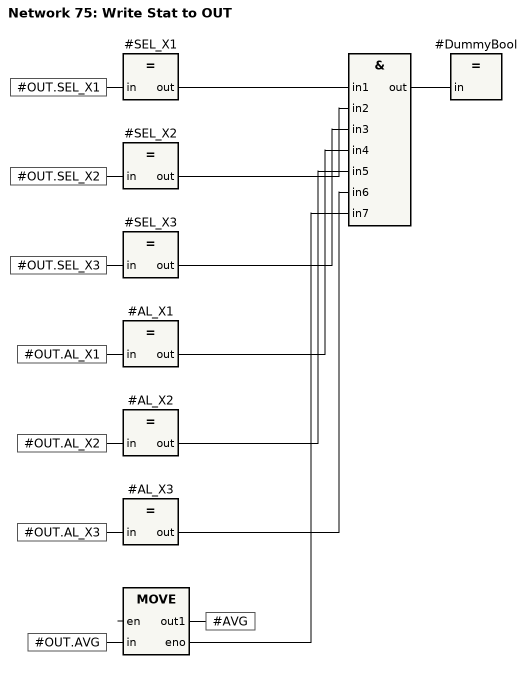
   #SEL_X1 := #OUT.SEL_X1;
   #SEL_X2 := #OUT.SEL_X2;
   #SEL_X3 := #OUT.SEL_X3;
   #AL_X1 := #OUT.AL_X1;
   #AL_X2 := #OUT.AL_X2;
   #AL_X3 := #OUT.AL_X3;
   #AVG := #OUT.AVG;
   #DummyBool := #OUT.SEL_X1 AND #OUT.SEL_X2 AND #OUT.SEL_X3 AND #OUT.AL_X1 AND #OUT.AL_X2 AND #OUT.AL_X3;
END_REGION
END_FUNCTION_BLOCK

FUNCTION_BLOCK "ACESYS_RAMP"   // FB235, FBD
TITLE = ACESYS V8.0 - Build 001 - Ramp Analog Value
{ S7_Optimized_Access := 'FALSE' }
AUTHOR : FLSmidth
FAMILY : ACESYS
NAME : RAMP
VERSION : 8.0
   VAR_INPUT
      Cycle_Time : Int;   // Block Update Time
      SIG_IN : Real;   // Signal Input
      Ramp_Time_Up : Real;   // Ramp Up Time (ms)
      Ramp_Time_Down : Real;   // Ramp Down Time (ms)
      En_Ramp_Up : Bool;   // Enable Ramp Up
      En_Ramp_Down : Bool;   // Enable Ramp Up
   END_VAR
   VAR_OUTPUT
      SIG_OUT : Real;   // Signal Out
   END_VAR
   VAR
      BlockInfo : Struct
         Ace_Version : Int;   // Acesys Block Version Number
         Ace_BuildNo : Int;   // Acesys Block Build Number
         DB_Number : Int;   // Block Instance DB Number
      END_STRUCT;
      Delta_X_Down : Real;   // Number of scan to ramp down
      Delta_X_Up : Real;   // Number of scan to ramp up
      Delta_Y : Real;
      PV_New : Real;
      PV_ToBe : Real;
      ScanTime_Real : Real;
      OUT : Struct
         SIG_OUT : Real;
      END_STRUCT;
      RunTime_Mem : LReal;
      RunTime_RetVal : LReal;
      RunTime_Result : LReal;
   END_VAR
   VAR_TEMP
      Aon : Bool;   // Always ON
      Aoff : Bool;   // Always OFF
      DummyBool : Bool;   // Dummy Bool
      DummyReal : Real;   // Dummy Real
      ScanTime_DINT : DInt;
      SIG_OUT_Internal : Real;   // Signal Out Temp.
      Ramp_Time_Up_Internal : Real;   // Ramp Up Time (ms)
      Ramp_Time_Down_Internal : Real;   // Ramp Down Time (ms)
   END_VAR
   VAR_TEMP   // added for the SCL form of the ladder/FBD networks
      _w1 : Bool;
   END_VAR
BEGIN

REGION Network 1: Always ON
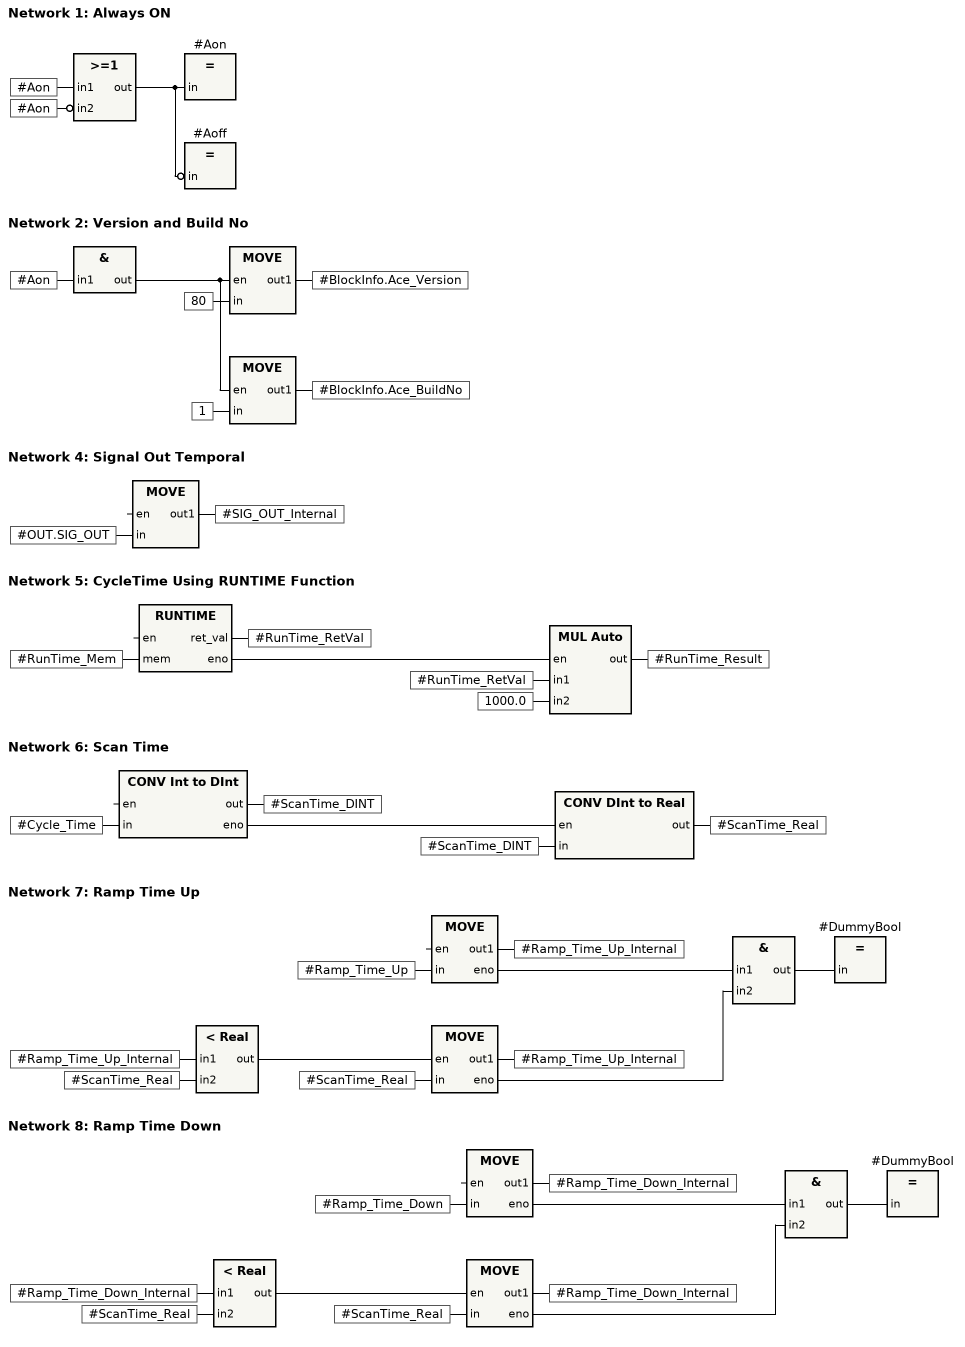
   #Aon := #Aon OR NOT #Aon;
   #Aoff := NOT #Aon;
END_REGION

REGION Network 2: Version and Build No
   IF #Aon THEN
       #BlockInfo.Ace_Version := 80;
       #BlockInfo.Ace_BuildNo := 1;
   END_IF;
END_REGION

REGION Network 3 (STL): Instance DB Number to Faceplate
         L     DINO;
         T     #BlockInfo.DB_Number;
END_REGION

REGION Network 4: Signal Out Temporal
   #SIG_OUT_Internal := #OUT.SIG_OUT;
END_REGION

REGION Network 5: CycleTime Using RUNTIME Function
   // no SCL statement known for Runtime: written as a call
   // ENO of a box is taken as its EN; it also drops when the box reports an error
   #RunTime_RetVal := Runtime(mem := #RunTime_Mem);
   #RunTime_Result := #RunTime_RetVal * 1000.0;
END_REGION

REGION Network 6: Scan Time
   // Build 2 - Cycle_Time added and defined as input to the block instead of MW110
   // ENO of a box is taken as its EN; it also drops when the box reports an error
   #ScanTime_DINT := INT_TO_DINT(#Cycle_Time);
   #ScanTime_Real := DINT_TO_REAL(#ScanTime_DINT);
END_REGION

REGION Network 7: Ramp Time Up
   #Ramp_Time_Up_Internal := #Ramp_Time_Up;
   #_w1 := #Ramp_Time_Up_Internal < #ScanTime_Real;
   IF #_w1 THEN #Ramp_Time_Up_Internal := #ScanTime_Real; END_IF;
   #DummyBool := #_w1;
END_REGION

REGION Network 8: Ramp Time Down
   #Ramp_Time_Down_Internal := #Ramp_Time_Down;
   #_w1 := #Ramp_Time_Down_Internal < #ScanTime_Real;
   IF #_w1 THEN #Ramp_Time_Down_Internal := #ScanTime_Real; END_IF;
   #DummyBool := #_w1;
END_REGION

REGION Network 9: Check for Start Ramping
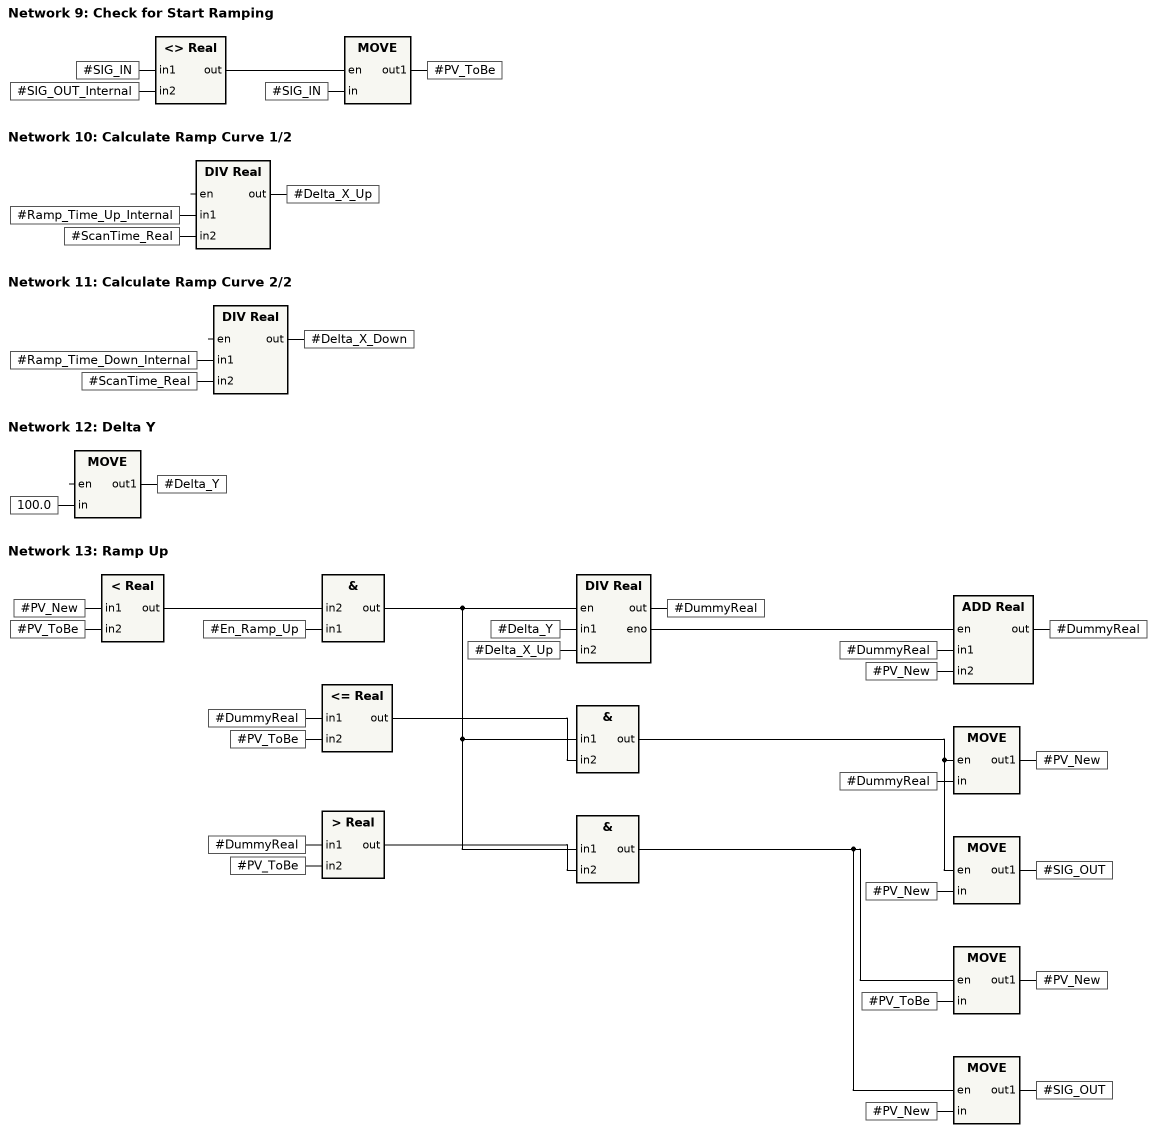
   IF #SIG_IN <> #SIG_OUT_Internal THEN #PV_ToBe := #SIG_IN; END_IF;
END_REGION

REGION Network 10: Calculate Ramp Curve 1/2
   #Delta_X_Up := #Ramp_Time_Up_Internal / #ScanTime_Real;
END_REGION

REGION Network 11: Calculate Ramp Curve 2/2
   #Delta_X_Down := #Ramp_Time_Down_Internal / #ScanTime_Real;
END_REGION

REGION Network 12: Delta Y
   #Delta_Y := 100.0;
END_REGION

REGION Network 13: Ramp Up
   // ENO of a box is taken as its EN; it also drops when the box reports an error
   #_w1 := (#PV_New < #PV_ToBe) AND #En_Ramp_Up;
   IF #_w1 THEN
       #DummyReal := #Delta_Y / #Delta_X_Up;
       #DummyReal := #DummyReal + #PV_New;
   END_IF;
   IF #_w1 AND (#DummyReal <= #PV_ToBe) THEN
       #PV_New := #DummyReal;
       #SIG_OUT := #PV_New;
   END_IF;
   IF #_w1 AND (#DummyReal > #PV_ToBe) THEN
       #PV_New := #PV_ToBe;
       #SIG_OUT := #PV_New;
   END_IF;
END_REGION

REGION Network 14: Ramp Down
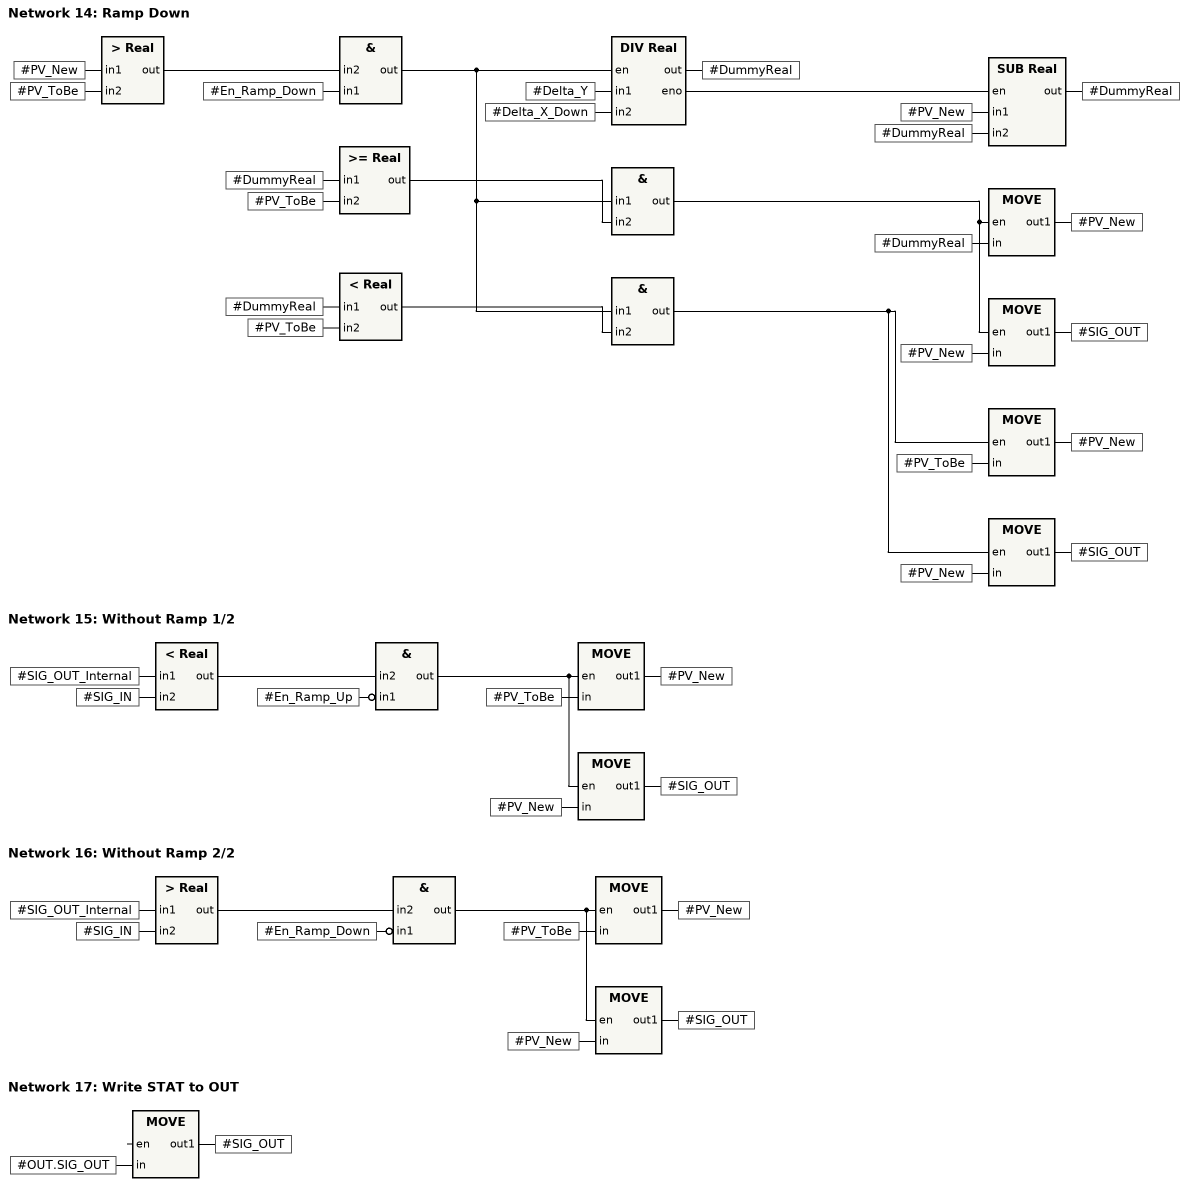
   // ENO of a box is taken as its EN; it also drops when the box reports an error
   #_w1 := (#PV_New > #PV_ToBe) AND #En_Ramp_Down;
   IF #_w1 THEN
       #DummyReal := #Delta_Y / #Delta_X_Down;
       #DummyReal := #PV_New - #DummyReal;
   END_IF;
   IF #_w1 AND (#DummyReal >= #PV_ToBe) THEN
       #PV_New := #DummyReal;
       #SIG_OUT := #PV_New;
   END_IF;
   IF #_w1 AND (#DummyReal < #PV_ToBe) THEN
       #PV_New := #PV_ToBe;
       #SIG_OUT := #PV_New;
   END_IF;
END_REGION

REGION Network 15: Without Ramp 1/2
   IF (#SIG_OUT_Internal < #SIG_IN) AND NOT #En_Ramp_Up THEN
       #PV_New := #PV_ToBe;
       #SIG_OUT := #PV_New;
   END_IF;
END_REGION

REGION Network 16: Without Ramp 2/2
   IF (#SIG_OUT_Internal > #SIG_IN) AND NOT #En_Ramp_Down THEN
       #PV_New := #PV_ToBe;
       #SIG_OUT := #PV_New;
   END_IF;
END_REGION

REGION Network 17: Write STAT to OUT
   #SIG_OUT := #OUT.SIG_OUT;
END_REGION
END_FUNCTION_BLOCK

FUNCTION_BLOCK "ACESTS_RPM"   // FB236, FBD
TITLE = ACESYS V8.0 - Build 005 - RPM Calculation
{ S7_Optimized_Access := 'FALSE' }
AUTHOR : FLSmidth
FAMILY : ACESYS
NAME : RPM
VERSION : 8.0
// Build 003 - Move all elements from TEMP to STAT Area
// Build 004 - RPM_Time Move issue  P_Trig  Placed to last 
// Build 005 - 07 Jan 2021 - Instead of using TIA Runtime Block replaced with Cycle Time Input
   VAR_INPUT
      Cycle_Time : Int;   // Block Update Time
      START : Bool;   // Unit Running
      EN_PULS : Bool;   // Enable Puls Signal
      EN_FREQ : Bool;   // Enable Process Input Signal
      PULS : Bool;   // Puls input
      FREQ : Real;   // Frequence input
      MAX_RPM : Real := 120.0;   // Max RPM (Used to calculate PCT)
      PULS_TURN : Int;   // Puls pr. Revolution
   END_VAR
   VAR_OUTPUT
      OUT_RPM : Real;   // Actual RPM
      OUT_PCT : Real;   // Actual RPM in %
   END_VAR
   VAR
      BlockInfo : Struct
         Ace_Version : Int;   // Acesys Block Version Number
         Ace_BuildNo : Int;   // Acesys Block Build Number
         DB_Number : Int;   // Block Instance DB Number
      END_STRUCT;
      ONS : Struct
         Pulse : Bool;
      END_STRUCT;
      Puls_Turn_Real : Real;
      Max_RPM_Internal : Real;
      PulseTimerAcc : Real;
      RPM_Time : Real;
      OUT_RPM_Temp_1 : Real;
      Out_PCT_Temp_1 : Real;
      TimerAcc : LReal;
      Time_Temp_1 : Int;
      Puls_Turn_Internal : DInt;
      Aon : Bool;
      Aoff : Bool;
      RPM_Pulse : Bool;
      EN_PULS_Temp : Bool;
      EN_FREQ_temp : Bool;
      RunTime_mem : LReal;
      RunTime_RetVal : LReal;
      RunTime_RetVal_Blk : LReal;
      RunTime_Result : LReal;
      OUT : Struct
         OUT_RPM : Real;
         OUT_PCT : Real;
      END_STRUCT;
   END_VAR
   VAR_TEMP
      DummyBool : Bool;
   END_VAR
   VAR_TEMP   // added for the SCL form of the ladder/FBD networks
      _w1 : Bool;
      _w2 : Bool;
   END_VAR
BEGIN

REGION Network 1: Always ON
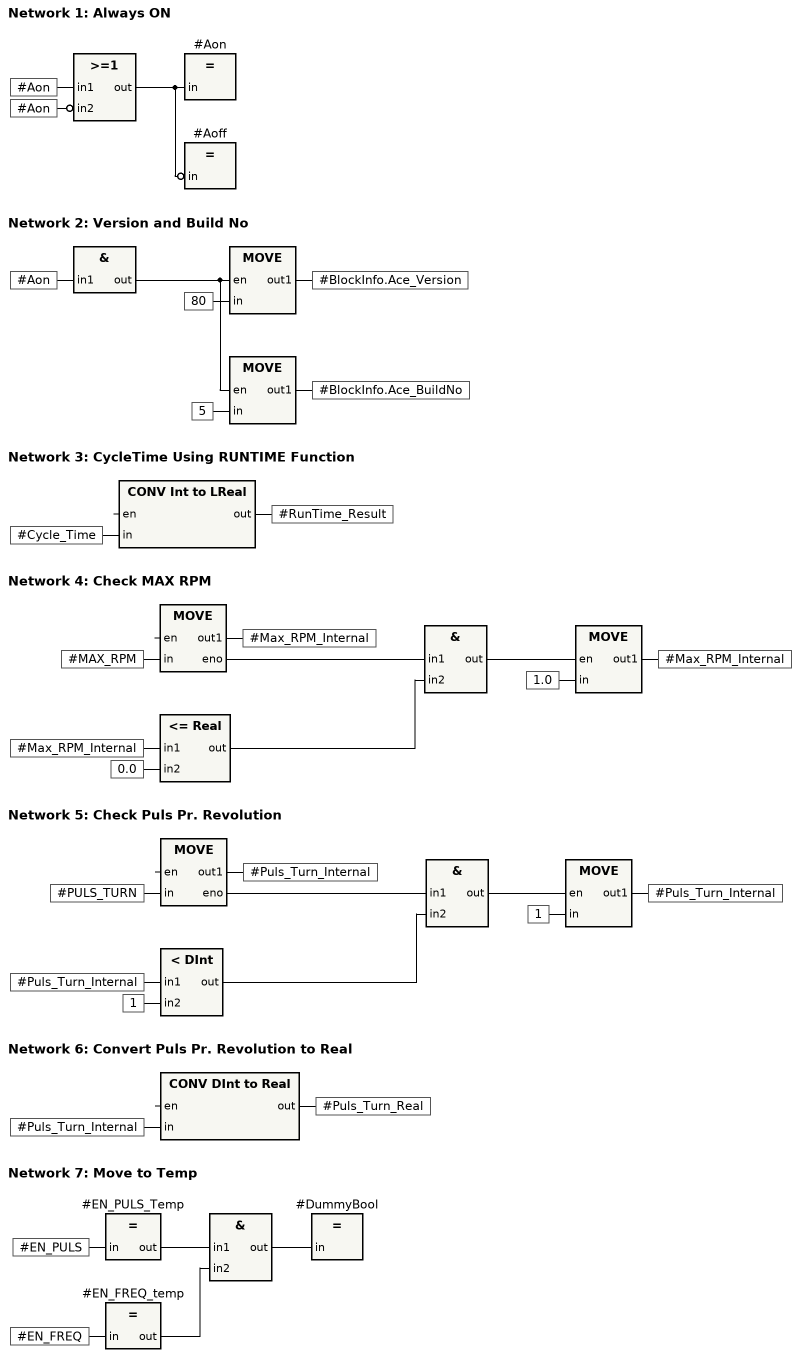
   #Aon := #Aon OR NOT #Aon;
   #Aoff := NOT #Aon;
END_REGION

REGION Network 2: Version and Build No
   IF #Aon THEN
       #BlockInfo.Ace_Version := 80;
       #BlockInfo.Ace_BuildNo := 5;
   END_IF;
END_REGION

REGION Network 3: CycleTime Using RUNTIME Function
   // Build 003 - 27 March 2019 - Use Runtime_RetVal_Blk of second runtime block to accurately get last scan time
   // Build 005 - 07 Jan 2021 - Instead of using TIA Runtime Block Output replaced with Cycle Time Input
   #RunTime_Result := INT_TO_LREAL(#Cycle_Time);
END_REGION

REGION Network 4: Check MAX RPM
   // ENO of a box is taken as its EN; it also drops when the box reports an error
   #Max_RPM_Internal := #MAX_RPM;
   IF #Max_RPM_Internal <= 0.0 THEN #Max_RPM_Internal := 1.0; END_IF;
END_REGION

REGION Network 5: Check Puls Pr. Revolution
   // ENO of a box is taken as its EN; it also drops when the box reports an error
   #Puls_Turn_Internal := #PULS_TURN;
   IF #Puls_Turn_Internal < 1 THEN #Puls_Turn_Internal := 1; END_IF;
END_REGION

REGION Network 6: Convert Puls Pr. Revolution to Real
   #Puls_Turn_Real := DINT_TO_REAL(#Puls_Turn_Internal);
END_REGION

REGION Network 7: Move to Temp
   #EN_PULS_Temp := #EN_PULS;
   #EN_FREQ_temp := #EN_FREQ;
   #DummyBool := #EN_PULS AND #EN_FREQ;
END_REGION

REGION Network 8: Check Configuration
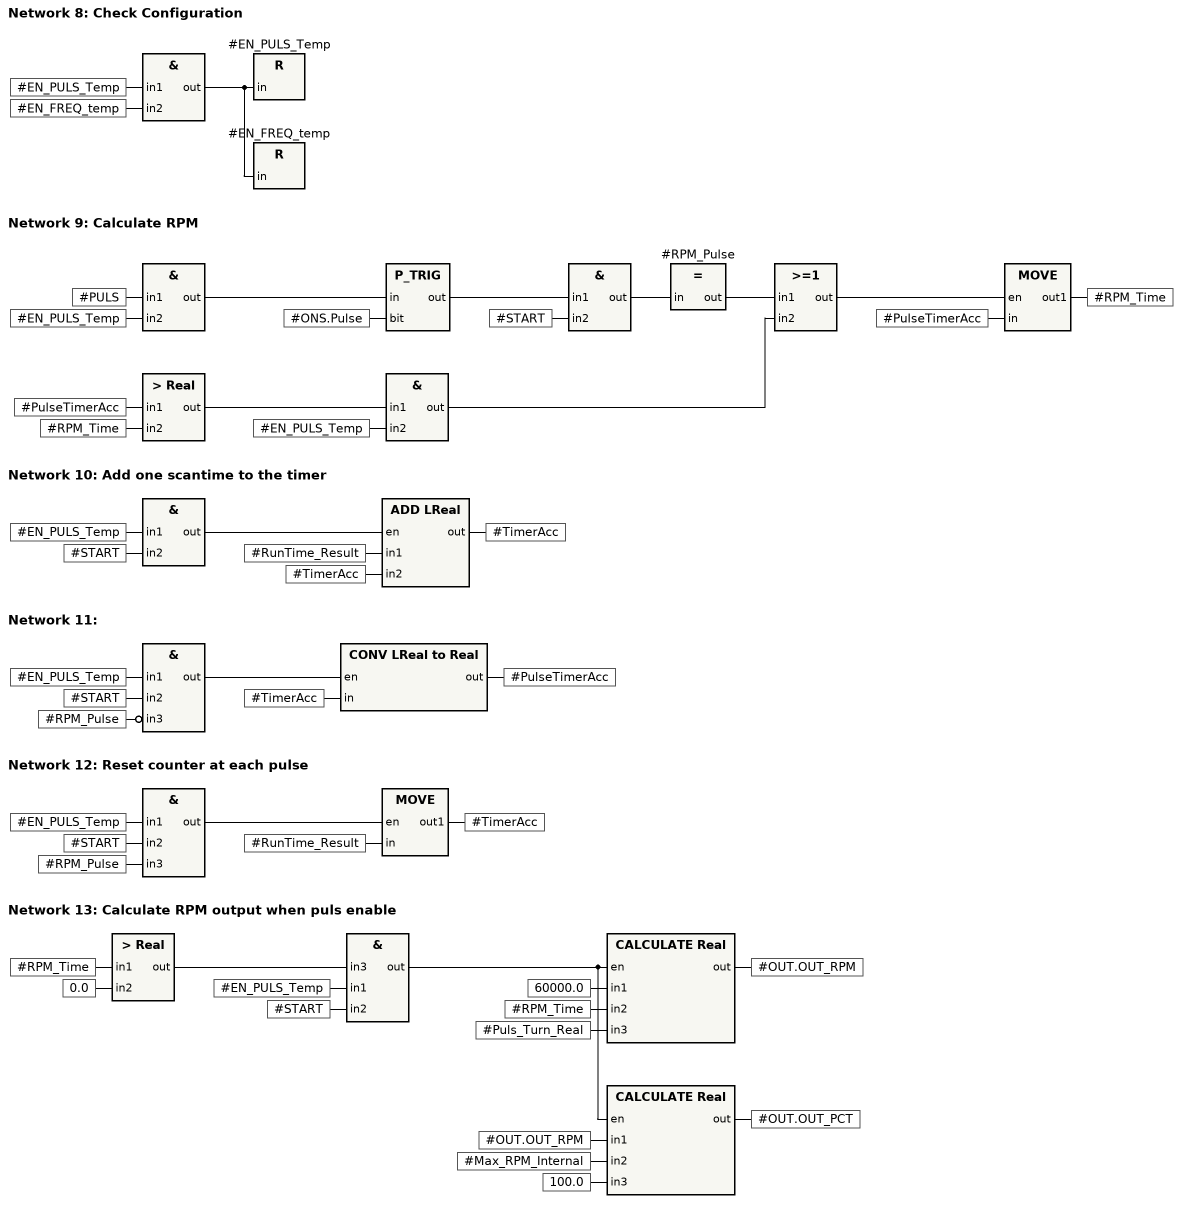
   #_w1 := #EN_PULS_Temp AND #EN_FREQ_temp;
   IF #_w1 THEN
       #EN_PULS_Temp := FALSE;
       #EN_FREQ_temp := FALSE;
   END_IF;
END_REGION

REGION Network 9: Calculate RPM
   // Calculate When a puls or when the time is longer than last Time
   // Build 004 - RPM_Time Move issue - P_Trig  Positioned last
   #_w1 := #PULS AND #EN_PULS_Temp;
   #_w2 := #_w1 AND NOT #ONS.Pulse;   // rising edge
   #ONS.Pulse := #_w1;
   #RPM_Pulse := #_w2 AND #START;
   IF #RPM_Pulse OR ((#PulseTimerAcc > #RPM_Time) AND #EN_PULS_Temp) THEN
       #RPM_Time := #PulseTimerAcc;
   END_IF;
END_REGION

REGION Network 10: Add one scantime to the timer
   // Build 003 - 27 March 2019 - Replace CycleTIme with Runtime_Result for internal Scan time of FB
   IF #EN_PULS_Temp AND #START THEN #TimerAcc := #RunTime_Result + #TimerAcc; END_IF;
END_REGION

REGION Network 11
   IF #EN_PULS_Temp AND #START AND NOT #RPM_Pulse THEN #PulseTimerAcc := LREAL_TO_REAL(#TimerAcc); END_IF;
END_REGION

REGION Network 12: Reset counter at each pulse
   // Build 003 - 27 March 2019 - Replace CycleTIme with Runtime_Result for internal Scan time of FB
   IF #EN_PULS_Temp AND #START AND #RPM_Pulse THEN #TimerAcc := #RunTime_Result; END_IF;
END_REGION

REGION Network 13: Calculate RPM output when puls enable
   // Build 005 - Average PCT Logic Typo Recified,Added 100.0 as IN3
   IF (#RPM_Time > 0.0) AND #EN_PULS_Temp AND #START THEN
       #OUT.OUT_RPM := (60000.0/#RPM_Time/#Puls_Turn_Real);
       #OUT.OUT_PCT := (#OUT.OUT_RPM/#Max_RPM_Internal)*100.0;
   END_IF;
END_REGION

REGION Network 14: Calculate RPM (Analog)
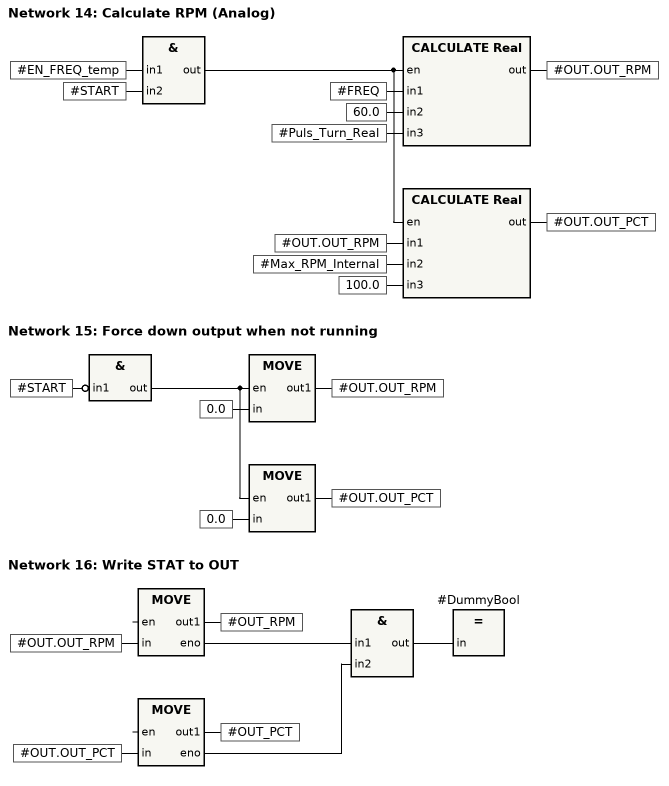
   IF #EN_FREQ_temp AND #START THEN
       #OUT.OUT_RPM := (#FREQ*60.0)/#Puls_Turn_Real;
       #OUT.OUT_PCT := (#OUT.OUT_RPM/#Max_RPM_Internal)*100.0;
   END_IF;
END_REGION

REGION Network 15: Force down output when not running
   IF NOT #START THEN
       #OUT.OUT_RPM := 0.0;
       #OUT.OUT_PCT := 0.0;
   END_IF;
END_REGION

REGION Network 16: Write STAT to OUT
   #OUT_RPM := #OUT.OUT_RPM;
   #OUT_PCT := #OUT.OUT_PCT;
   #DummyBool := TRUE;
END_REGION

REGION Network 17: Runtime Calculation of the block
   // Build 003 - 27 March 2019 - New Network - Runtime Block added to last network to accurately read FB execution time
   // Build 005 - 07 Jan 2021 - TIA Runtime Instruction deleted, Replace with Cycle Time Input
END_REGION
END_FUNCTION_BLOCK

FUNCTION_BLOCK "ACESYS_POWER"   // FB237, FBD
TITLE = ACESYS V8.0 - Build 001 - POWER MONITORING
{ S7_Optimized_Access := 'FALSE' }
AUTHOR : FLSmidth
FAMILY : ACESYS
NAME : POWER
VERSION : 8.0
   VAR_INPUT
      AL_SUPR : Bool;   // Alarm Supress by Program
   END_VAR
   VAR_OUTPUT
      MSW : "ACESYS_HMI_STAT_32T";
   END_VAR
   VAR_IN_OUT
      TOKEN : "ACESYS_TOKEN";
   END_VAR
   VAR
      BlockInfo : Struct
         Ace_Version : Int;   // Acesys Block Version Number
         Ace_BuildNo : Int;   // Acesys Block Build Number
         DB_Number : Int;   // Block Instance DB Number
      END_STRUCT;
      FP_CMD : Struct
         Spare_08 : Bool;
         Spare_09 : Bool;
         Spare_10 : Bool;
         Spare_11 : Bool;
         Spare_12 : Bool;
         Spare_13 : Bool;
         Spare_14 : Bool;
         AckAlarm : Bool;
         Reset : Bool;
         Spare_01 : Bool;
         Spare_02 : Bool;
         Spare_03 : Bool;
         Spare_04 : Bool;
         Spare_05 : Bool;
         Spare_06 : Bool;
         Spare_07 : Bool;
      END_STRUCT;
      FP_SEL : Struct
         Spare_08 : Bool;
         Spare_09 : Bool;
         Spare_10 : Bool;
         Spare_11 : Bool;
         Spare_12 : Bool;
         Spare_13 : Bool;
         Spare_14 : Bool;
         Spare_15 : Bool;
         Type_Monitor : Bool;
         Type_MVfeeder : Bool;
         Type_MVmotor : Bool;
         Type_NotSelected : Bool;
         ParentSupress : Bool;
         ParentSupressUnit : Bool;
         Spare_06 : Bool;
         Spare_07 : Bool;
      END_STRUCT;
      FP_SHOW : Struct
         VOLT_LNPH : Bool;   // Phase to pahse & Line to Neutral Voltage V/kV)
         CURR_LN : Bool;   // Line Current
         APOW_PH : Bool;   // Phase Power kW/MW)
         FRQ : Bool;   // Frequency (Hz)
         APOW_AVG : Bool;   // Average Apparent Power (kVA/MVA)
         RTPOW_AVG : Bool;   // Average Reactive Power (kW/MW)
         VOLT_UNBAL : Bool;   // Voltage Unbalance (%)
         CURR_UNBAL : Bool;   // Current unbalance (%)
         VOLT_THD : Bool;   // Total Hormonic Distorsion Voltage (%)
         CURR_THD : Bool;   // Total Hormonic Distorsion Current (%)
         RENG : Bool;   // Average Reactive Energy (kVARH/MVARH)
         kWH_REV : Bool;   // Reverse kWH (kWhr/MWhr)
         kVAH_FwdRev : Bool;   // kVAH Forward/Reverse(kVAH/MVAH)
         kVARH_Rev : Bool;   // kVARH Reverse(kVARH/MVARH)
         MD_kW_Fwd : Bool;   // kW Forward (kW/MW)
         MD_kW_Rev : Bool;   // kW Reverse (kW/MW)
         MD_kVAr_Fwd : Bool;   // kVA Forward (kVAr/MVAr)
         MD_kVAr_Rev : Bool;   // kVA Reverse (kVAr/MVAr)
         HORM_5TH : Bool;   // 5th Order Hormonics
         HORM_7TH : Bool;   // 7th Order Hormonics
         HORM_11TH : Bool;   // 11th Order Hormonics
         MWT : Bool;   // Motor Winding temperature
         MBT : Bool;   // Motor Bearing temperature
         TWT : Bool;   // Transformer Winding temperature
         TOT : Bool;   // Transformer Oil temperature
         RunHrs : Bool;   // Run Hours
         PB_Reset : Bool;
         PQ2 : Bool;   // Power Quality 2 Group Box
         Temperature : Bool;   // Power Group Box
         Spare19 : Bool;   // Energy Group Box
         Spare18 : Bool;
         Spare17 : Bool;
         Spare16 : Bool;
         Spare15 : Bool;
         Spare14 : Bool;
         Spare13 : Bool;
         Spare12 : Bool;
         Spare11 : Bool;
         Spare10 : Bool;
         Spare09 : Bool;
         Spare08 : Bool;
         Spare07 : Bool;
         Spare06 : Bool;
         Spare05 : Bool;
         Spare04 : Bool;
         Spare03 : Bool;
         Spare02 : Bool;
         Spare01 : Bool;
      END_STRUCT;
      FP_VIS : Struct
         VOLT_LNPH : Bool;   // Phase to pahse & Line to Neutral Voltage V/kV)
         CURR_LN : Bool;   // Line Current
         APOW_PH : Bool;   // Phase Power kW/MW)
         FRQ : Bool;   // Frequency (Hz)
         APOW_AVG : Bool;   // Average Apparent Power (kVA/MVA)
         RTPOW_AVG : Bool;   // Average Reactive Power (kW/MW)
         VOLT_UNBAL : Bool;   // Voltage Unbalance (%)
         CURR_UNBAL : Bool;   // Current unbalance (%)
         VOLT_THD : Bool;   // Total Hormonic Distorsion Voltage (%)
         CURR_THD : Bool;   // Total Hormonic Distorsion Current (%)
         RENG : Bool;   // Average Reactive Energy (kVARH/MVARH)
         kWH_REV : Bool;   // Reverse kWH (kWhr/MWhr)
         kVAH_FwdRev : Bool;   // kVAH Forward/Reverse(kVAH/MVAH)
         kVARH_Rev : Bool;   // kVARH Reverse(kVARH/MVARH)
         MD_kW_Fwd : Bool;   // kW Forward (kW/MW)
         MD_kW_Rev : Bool;   // kW Reverse (kW/MW)
         MD_kVAr_Fwd : Bool;   // kVA Forward (kVAr/MVAr)
         MD_kVAr_Rev : Bool;   // kVA Reverse (kVAr/MVAr)
         HORM_5TH : Bool;   // 5th Order Hormonics
         HORM_7TH : Bool;   // 7th Order Hormonics
         HORM_11TH : Bool;   // 11th Order Hormonics
         MWT : Bool;   // Motor Winding temperature
         MBT : Bool;   // Motor Bearing temperature
         TWT : Bool;   // Transformer Winding temperature
         TOT : Bool;   // Transformer Oil temperature
         RunHrs : Bool;   // Run Hours
         PB_Reset : Bool;   // Show Push Button Reset
         PQ2 : Bool;   // Power Quality 2 Group Box
         Power : Bool;   // Power Group Box
         Energy : Bool;   // Energy Group Box
         Temperature : Bool;
         Spare17 : Bool;
         Spare16 : Bool;
         Spare15 : Bool;
         Spare14 : Bool;
         Spare13 : Bool;
         Spare12 : Bool;
         Spare11 : Bool;
         Spare10 : Bool;
         Spare09 : Bool;
         Spare08 : Bool;
         Spare07 : Bool;
         Spare06 : Bool;
         Spare05 : Bool;
         Spare04 : Bool;
         Spare03 : Bool;
         Spare02 : Bool;
         Spare01 : Bool;
      END_STRUCT;
      LINK : "ACESYS_PowerLink";
      Volt_L1N : Real;   // R Phase to Neutral Voltage Calc
      Volt_L2N : Real;   // Y Phase to Neutral Voltage Calc
      Volt_L3N : Real;   // B Phase to Neutral Voltage Calc
      ONS : Struct
         Spare_08 : Bool;
         Spare_09 : Bool;
         Spare_10 : Bool;
         Spare_11 : Bool;
         Spare_12 : Bool;
         Spare_13 : Bool;
         Spare_14 : Bool;
         Spare_15 : Bool;
         AckAlarm : Bool;
         Spare_01 : Bool;
         Spare_02 : Bool;
         Spare_03 : Bool;
         Spare_04 : Bool;
         Spare_05 : Bool;
         Spare_06 : Bool;
         Spare_07 : Bool;
      END_STRUCT;
      StatusWork : Int;
      AlarmNo : Int;
      AlarmNo_Old : Int;
      CMD_Reset : Bool;
      CMD_AckAlarm : Bool;
      ALARM_SupressionActive : Bool;
      ALARM_AlarmPresent : Bool;
      ALARM_FailureAckRequired : Bool;
      FPCMD_RESET_TMR : TON_TIME;
      MSW_Status_Trans : Int;
   END_VAR
   VAR_TEMP
      ADAPT_Pntr : Struct
         DB_Number : Word;
         Offset_Address : DWord;
      END_STRUCT;
      Aon : Bool;
      Aoff : Bool;
      DummyBool : Bool;
      DummyInt : Int;
      DummyDInt : DInt;
      Temp_AR1 : DWord;
      TEMP_AR2 : DWord;
      Offset : DWord;
      Pntr_ADAPT : ANY;
      Pntr_ADAPT_LC : ANY;
      Pntr_DATA : ANY;
      Pntr_ADAPT_Source : ANY;
   END_VAR
   VAR_TEMP   // added for the SCL form of the ladder/FBD networks
      _w1 : Bool;
   END_VAR
BEGIN

REGION Network 1: Always ON
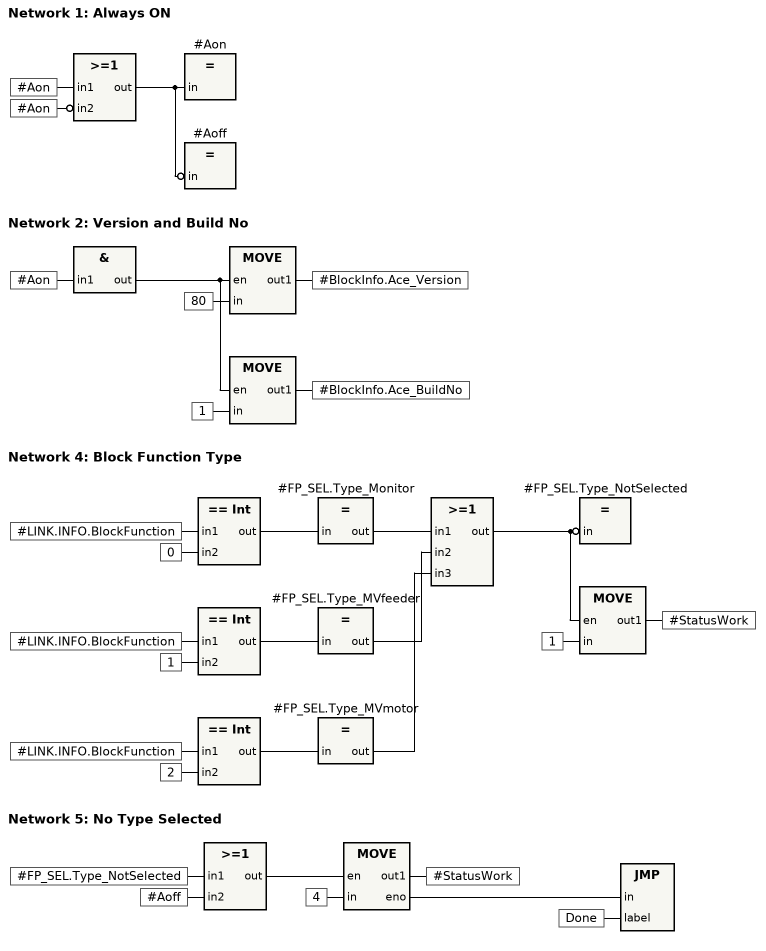
   #Aon := #Aon OR NOT #Aon;
   #Aoff := NOT #Aon;
END_REGION

REGION Network 2: Version and Build No
   IF #Aon THEN
       #BlockInfo.Ace_Version := 80;
       #BlockInfo.Ace_BuildNo := 1;
   END_IF;
END_REGION

REGION Network 3 (STL): Instance DB Number to Faceplate
         L     DINO;
         T     #BlockInfo.DB_Number;
END_REGION

REGION Network 4: Block Function Type
   #FP_SEL.Type_Monitor := #LINK.INFO.BlockFunction = 0;
   #FP_SEL.Type_MVfeeder := #LINK.INFO.BlockFunction = 1;
   #FP_SEL.Type_MVmotor := #LINK.INFO.BlockFunction = 2;
   #_w1 := #FP_SEL.Type_Monitor OR #FP_SEL.Type_MVfeeder OR #FP_SEL.Type_MVmotor;
   #FP_SEL.Type_NotSelected := NOT #_w1;
   IF #_w1 THEN #StatusWork := 1; END_IF;
END_REGION

REGION Network 5: No Type Selected
   // ENO of a box is taken as its EN; it also drops when the box reports an error
   #_w1 := #FP_SEL.Type_NotSelected OR #Aoff;
   IF #_w1 THEN
       #StatusWork := 4;
       GOTO Done;
   END_IF;
END_REGION

REGION Network 6: Set Show Parameters
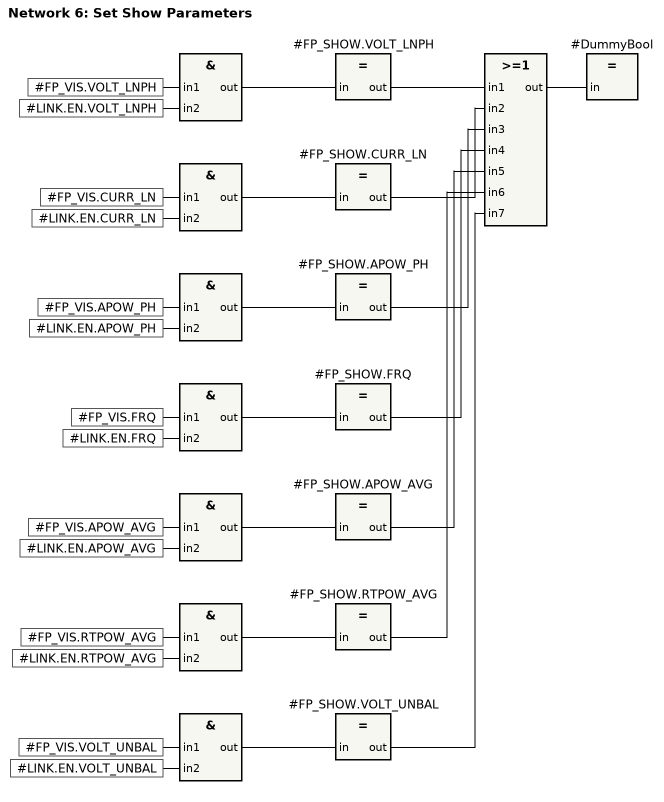
   #FP_SHOW.VOLT_LNPH := #FP_VIS.VOLT_LNPH AND #LINK.EN.VOLT_LNPH;
   #FP_SHOW.CURR_LN := #FP_VIS.CURR_LN AND #LINK.EN.CURR_LN;
   #FP_SHOW.APOW_PH := #FP_VIS.APOW_PH AND #LINK.EN.APOW_PH;
   #FP_SHOW.FRQ := #FP_VIS.FRQ AND #LINK.EN.FRQ;
   #FP_SHOW.APOW_AVG := #FP_VIS.APOW_AVG AND #LINK.EN.APOW_AVG;
   #FP_SHOW.RTPOW_AVG := #FP_VIS.RTPOW_AVG AND #LINK.EN.RTPOW_AVG;
   #FP_SHOW.VOLT_UNBAL := #FP_VIS.VOLT_UNBAL AND #LINK.EN.VOLT_UNBAL;
   #DummyBool := #FP_SHOW.VOLT_LNPH OR #FP_SHOW.CURR_LN OR #FP_SHOW.APOW_PH OR #FP_SHOW.FRQ OR #FP_SHOW.APOW_AVG OR #FP_SHOW.RTPOW_AVG OR #FP_SHOW.VOLT_UNBAL;
END_REGION

REGION Network 7: Set Show Parameters
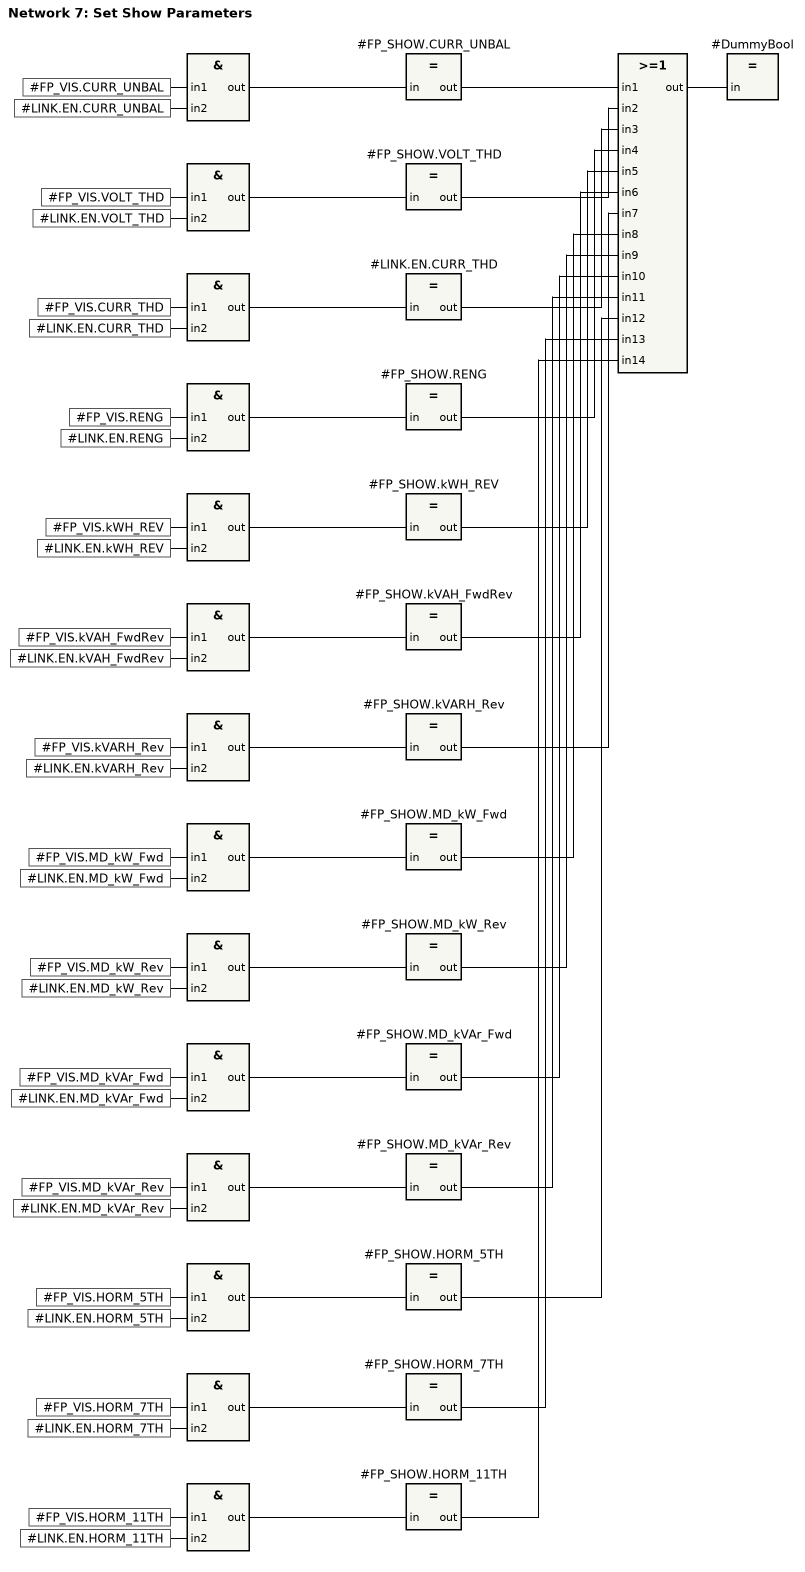
   #FP_SHOW.CURR_UNBAL := #FP_VIS.CURR_UNBAL AND #LINK.EN.CURR_UNBAL;
   #FP_SHOW.VOLT_THD := #FP_VIS.VOLT_THD AND #LINK.EN.VOLT_THD;
   #LINK.EN.CURR_THD := #FP_VIS.CURR_THD AND #LINK.EN.CURR_THD;
   #FP_SHOW.RENG := #FP_VIS.RENG AND #LINK.EN.RENG;
   #FP_SHOW.kWH_REV := #FP_VIS.kWH_REV AND #LINK.EN.kWH_REV;
   #FP_SHOW.kVAH_FwdRev := #FP_VIS.kVAH_FwdRev AND #LINK.EN.kVAH_FwdRev;
   #FP_SHOW.kVARH_Rev := #FP_VIS.kVARH_Rev AND #LINK.EN.kVARH_Rev;
   #FP_SHOW.MD_kW_Fwd := #FP_VIS.MD_kW_Fwd AND #LINK.EN.MD_kW_Fwd;
   #FP_SHOW.MD_kW_Rev := #FP_VIS.MD_kW_Rev AND #LINK.EN.MD_kW_Rev;
   #FP_SHOW.MD_kVAr_Fwd := #FP_VIS.MD_kVAr_Fwd AND #LINK.EN.MD_kVAr_Fwd;
   #FP_SHOW.MD_kVAr_Rev := #FP_VIS.MD_kVAr_Rev AND #LINK.EN.MD_kVAr_Rev;
   #FP_SHOW.HORM_5TH := #FP_VIS.HORM_5TH AND #LINK.EN.HORM_5TH;
   #FP_SHOW.HORM_7TH := #FP_VIS.HORM_7TH AND #LINK.EN.HORM_7TH;
   #FP_SHOW.HORM_11TH := #FP_VIS.HORM_11TH AND #LINK.EN.HORM_11TH;
   #DummyBool := #FP_SHOW.CURR_UNBAL OR #FP_SHOW.VOLT_THD OR #LINK.EN.CURR_THD OR #FP_SHOW.RENG OR #FP_SHOW.kWH_REV OR #FP_SHOW.kVAH_FwdRev OR #FP_SHOW.kVARH_Rev OR #FP_SHOW.MD_kW_Fwd OR #FP_SHOW.MD_kW_Rev OR #FP_SHOW.MD_kVAr_Fwd OR #FP_SHOW.MD_kVAr_Rev OR #FP_SHOW.HORM_5TH OR #FP_SHOW.HORM_7TH OR #FP_SHOW.HORM_11TH;
END_REGION

REGION Network 8: Set Show Parameters
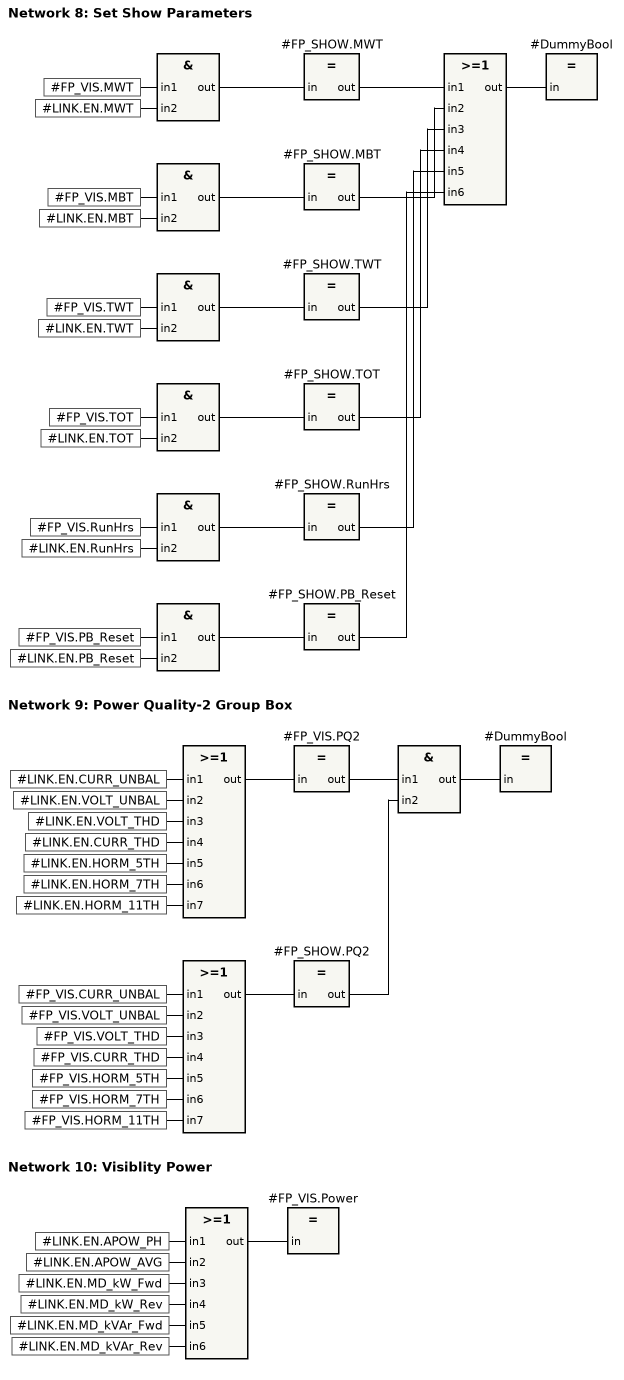
   #FP_SHOW.MWT := #FP_VIS.MWT AND #LINK.EN.MWT;
   #FP_SHOW.MBT := #FP_VIS.MBT AND #LINK.EN.MBT;
   #FP_SHOW.TWT := #FP_VIS.TWT AND #LINK.EN.TWT;
   #FP_SHOW.TOT := #FP_VIS.TOT AND #LINK.EN.TOT;
   #FP_SHOW.RunHrs := #FP_VIS.RunHrs AND #LINK.EN.RunHrs;
   #FP_SHOW.PB_Reset := #FP_VIS.PB_Reset AND #LINK.EN.PB_Reset;
   #DummyBool := #FP_SHOW.MWT OR #FP_SHOW.MBT OR #FP_SHOW.TWT OR #FP_SHOW.TOT OR #FP_SHOW.RunHrs OR #FP_SHOW.PB_Reset;
END_REGION

REGION Network 9: Power Quality-2 Group Box
   #FP_VIS.PQ2 := #LINK.EN.CURR_UNBAL OR #LINK.EN.VOLT_UNBAL OR #LINK.EN.VOLT_THD OR #LINK.EN.CURR_THD OR #LINK.EN.HORM_5TH OR #LINK.EN.HORM_7TH OR #LINK.EN.HORM_11TH;
   #FP_SHOW.PQ2 := #FP_VIS.CURR_UNBAL OR #FP_VIS.VOLT_UNBAL OR #FP_VIS.VOLT_THD OR #FP_VIS.CURR_THD OR #FP_VIS.HORM_5TH OR #FP_VIS.HORM_7TH OR #FP_VIS.HORM_11TH;
   #DummyBool := #FP_VIS.PQ2 AND #FP_SHOW.PQ2;
END_REGION

REGION Network 10: Visiblity Power
   #FP_VIS.Power := #LINK.EN.APOW_PH OR #LINK.EN.APOW_AVG OR #LINK.EN.MD_kW_Fwd OR #LINK.EN.MD_kW_Rev OR #LINK.EN.MD_kVAr_Fwd OR #LINK.EN.MD_kVAr_Rev;
END_REGION

REGION Network 11: Visiblity Energy
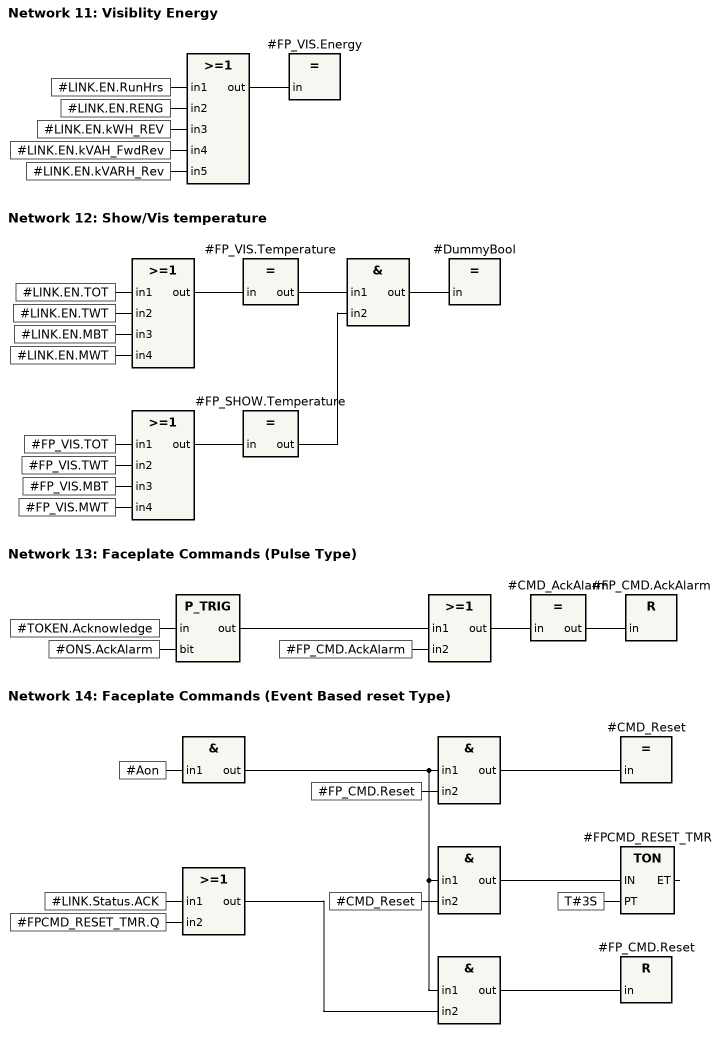
   #FP_VIS.Energy := #LINK.EN.RunHrs OR #LINK.EN.RENG OR #LINK.EN.kWH_REV OR #LINK.EN.kVAH_FwdRev OR #LINK.EN.kVARH_Rev;
END_REGION

REGION Network 12: Show/Vis temperature
   #FP_VIS.Temperature := #LINK.EN.TOT OR #LINK.EN.TWT OR #LINK.EN.MBT OR #LINK.EN.MWT;
   #FP_SHOW.Temperature := #FP_VIS.TOT OR #FP_VIS.TWT OR #FP_VIS.MBT OR #FP_VIS.MWT;
   #DummyBool := #FP_VIS.Temperature AND #FP_SHOW.Temperature;
END_REGION

REGION Network 13: Faceplate Commands (Pulse Type)
   #_w1 := #TOKEN.Acknowledge AND NOT #ONS.AckAlarm;   // rising edge
   #ONS.AckAlarm := #TOKEN.Acknowledge;
   #CMD_AckAlarm := #_w1 OR #FP_CMD.AckAlarm;
   IF #CMD_AckAlarm THEN #FP_CMD.AckAlarm := FALSE; END_IF;
END_REGION

REGION Network 14: Faceplate Commands (Event Based reset Type)
   #CMD_Reset := #Aon AND #FP_CMD.Reset;
   #FPCMD_RESET_TMR(IN := #Aon AND #CMD_Reset, PT := T#3S);   // TON
   IF #Aon AND (#LINK.Status.ACK OR #FPCMD_RESET_TMR.Q) THEN #FP_CMD.Reset := FALSE; END_IF;
END_REGION

REGION Network 15: Phase to Neutral Voltage Calcuation
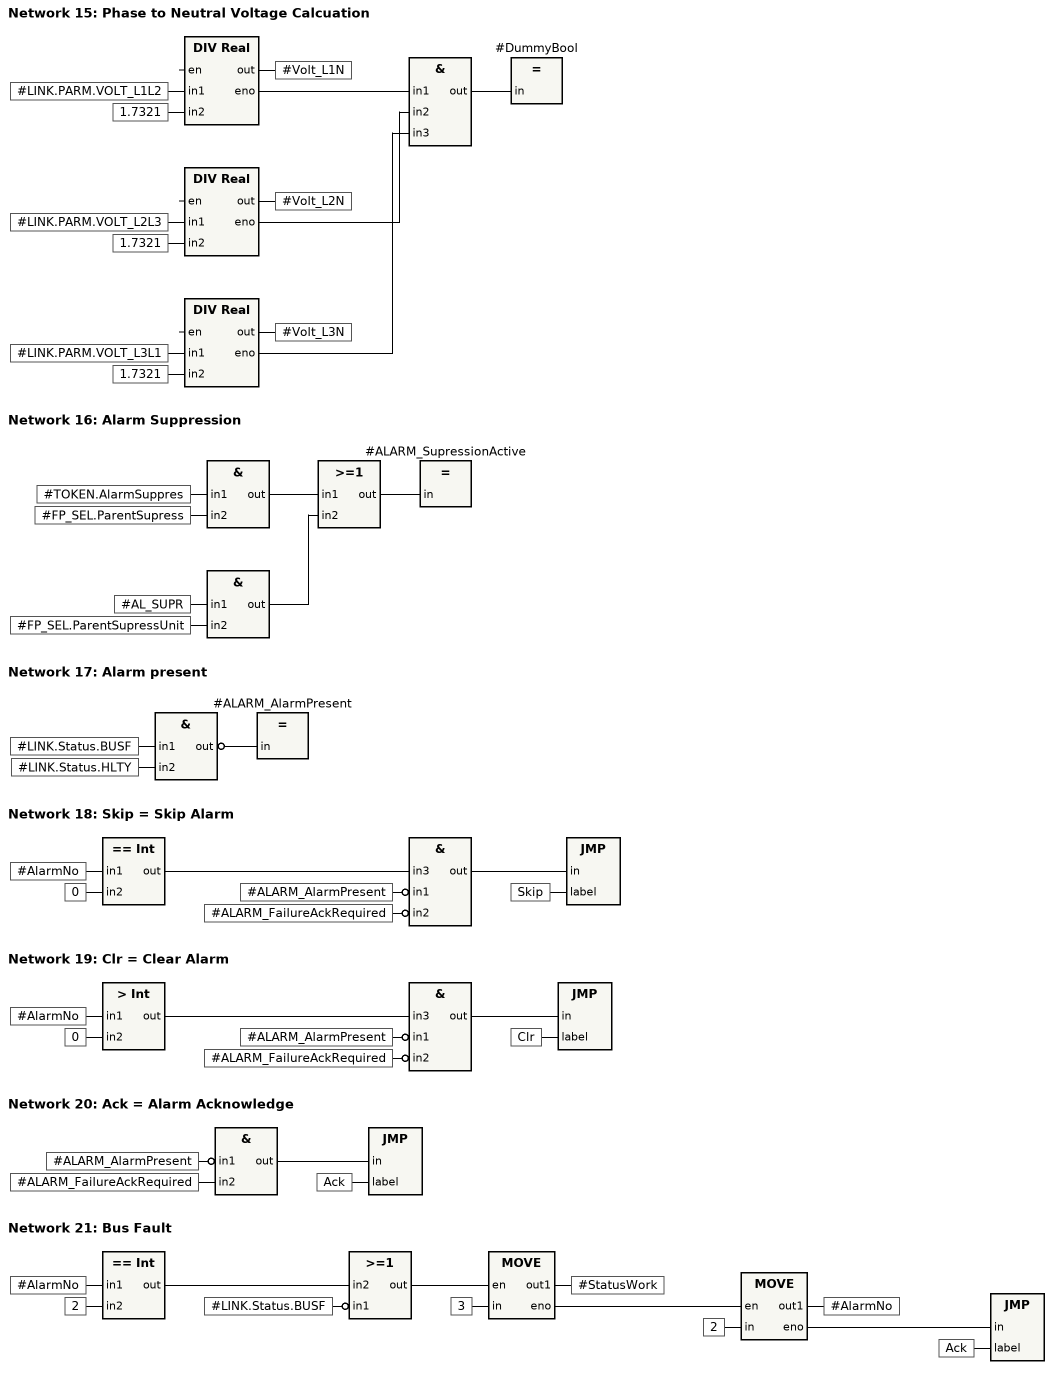
   // ENO of a box is taken as its EN; it also drops when the box reports an error
   #Volt_L1N := #LINK.PARM.VOLT_L1L2 / 1.7321;
   #Volt_L2N := #LINK.PARM.VOLT_L2L3 / 1.7321;
   #Volt_L3N := #LINK.PARM.VOLT_L3L1 / 1.7321;
   #DummyBool := TRUE;
END_REGION

REGION Network 16: Alarm Suppression
   #ALARM_SupressionActive := (#TOKEN.AlarmSuppres AND #FP_SEL.ParentSupress) OR (#AL_SUPR AND #FP_SEL.ParentSupressUnit);
END_REGION

REGION Network 17: Alarm present
   #ALARM_AlarmPresent := NOT (#LINK.Status.BUSF AND #LINK.Status.HLTY);
END_REGION

REGION Network 18: Skip = Skip Alarm
   IF (#AlarmNo = 0) AND NOT #ALARM_AlarmPresent AND NOT #ALARM_FailureAckRequired THEN GOTO Skip; END_IF;
END_REGION

REGION Network 19: Clr = Clear Alarm
   IF (#AlarmNo > 0) AND NOT #ALARM_AlarmPresent AND NOT #ALARM_FailureAckRequired THEN GOTO Clr; END_IF;
END_REGION

REGION Network 20: Ack = Alarm Acknowledge
   IF NOT #ALARM_AlarmPresent AND #ALARM_FailureAckRequired THEN GOTO Ack; END_IF;
END_REGION

REGION Network 21: Bus Fault
   // ENO of a box is taken as its EN; it also drops when the box reports an error
   #_w1 := (#AlarmNo = 2) OR NOT #LINK.Status.BUSF;
   IF #_w1 THEN
       #StatusWork := 3;
       #AlarmNo := 2;
       GOTO Ack;
   END_IF;
END_REGION

REGION Network 22: Device Healthy
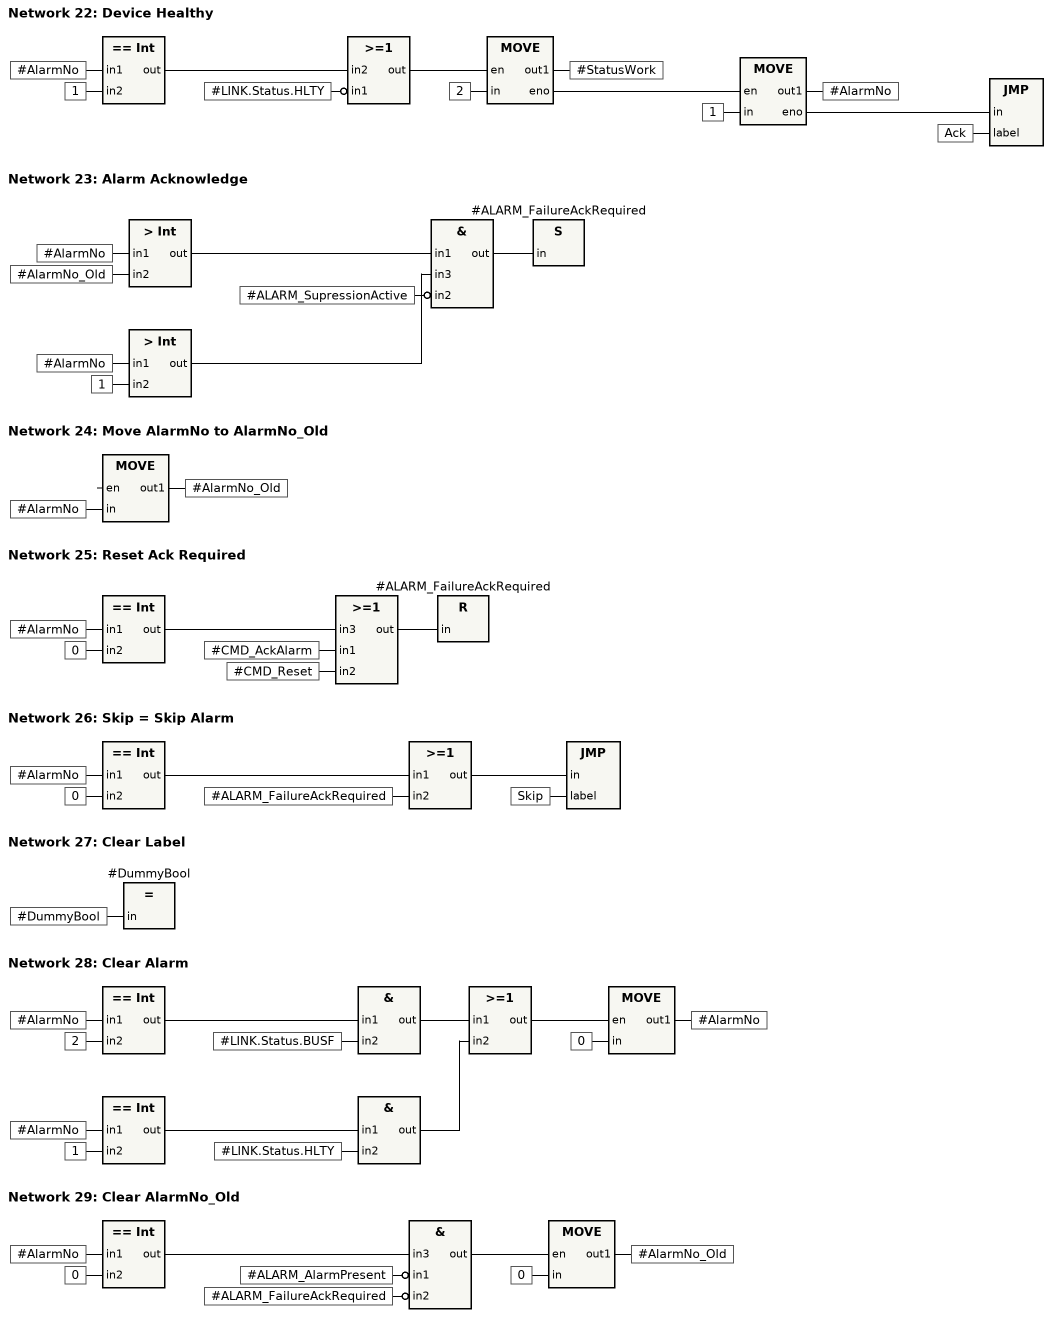
   // ENO of a box is taken as its EN; it also drops when the box reports an error
   #_w1 := (#AlarmNo = 1) OR NOT #LINK.Status.HLTY;
   IF #_w1 THEN
       #StatusWork := 2;
       #AlarmNo := 1;
       GOTO Ack;
   END_IF;
END_REGION

REGION Network 23: Alarm Acknowledge
   Ack:
   IF (#AlarmNo > #AlarmNo_Old) AND (#AlarmNo > 1) AND NOT #ALARM_SupressionActive THEN
       #ALARM_FailureAckRequired := TRUE;
   END_IF;
END_REGION

REGION Network 24: Move AlarmNo to AlarmNo_Old
   #AlarmNo_Old := #AlarmNo;
END_REGION

REGION Network 25: Reset Ack Required
   IF (#AlarmNo = 0) OR #CMD_AckAlarm OR #CMD_Reset THEN #ALARM_FailureAckRequired := FALSE; END_IF;
END_REGION

REGION Network 26: Skip = Skip Alarm
   IF (#AlarmNo = 0) OR #ALARM_FailureAckRequired THEN GOTO Skip; END_IF;
END_REGION

REGION Network 27: Clear Label
   Clr:
   #DummyBool := #DummyBool;
END_REGION

REGION Network 28: Clear Alarm
   IF ((#AlarmNo = 2) AND #LINK.Status.BUSF) OR ((#AlarmNo = 1) AND #LINK.Status.HLTY) THEN
       #AlarmNo := 0;
   END_IF;
END_REGION

REGION Network 29: Clear AlarmNo_Old
   IF (#AlarmNo = 0) AND NOT #ALARM_AlarmPresent AND NOT #ALARM_FailureAckRequired THEN
       #AlarmNo_Old := 0;
   END_IF;
END_REGION

REGION Network 30: Return if Skip Alarm
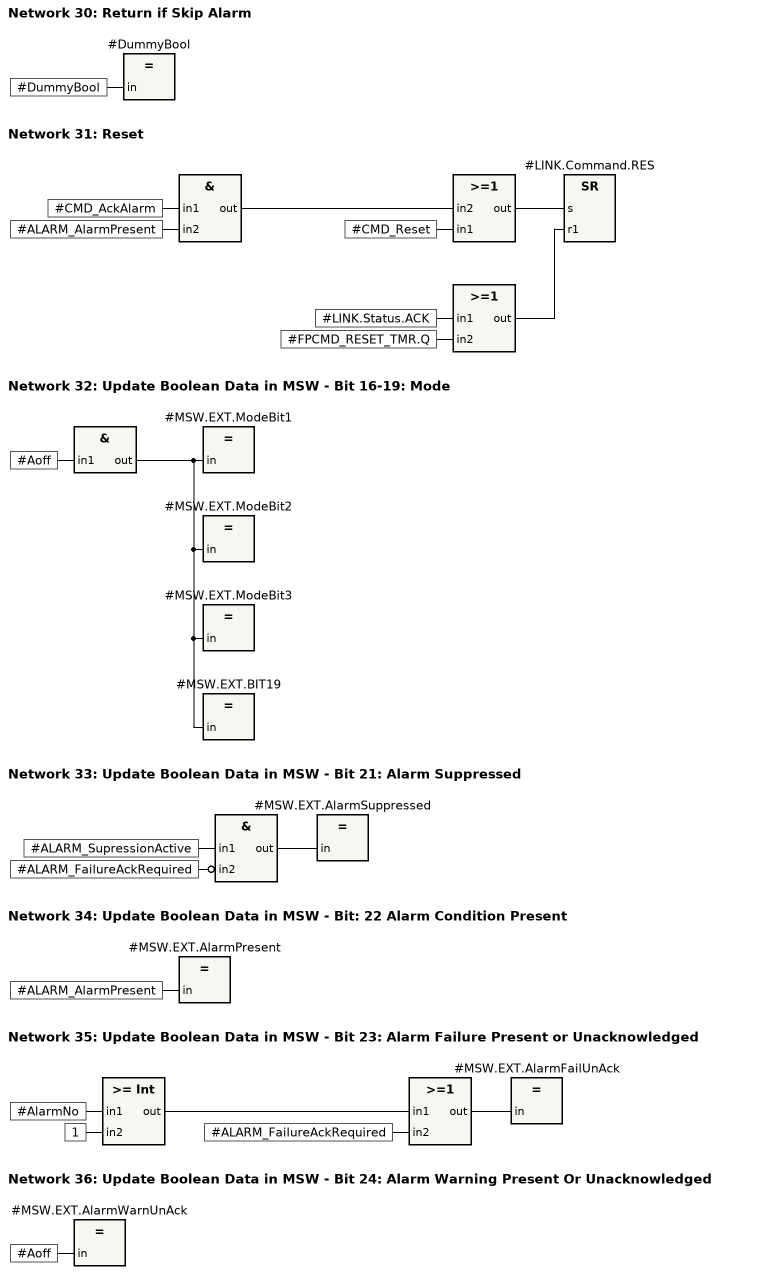
   Skip:
   #DummyBool := #DummyBool;
END_REGION

REGION Network 31: Reset
   IF (#CMD_AckAlarm AND #ALARM_AlarmPresent) OR #CMD_Reset THEN
       #LINK.Command.RES := TRUE;   // SR flip-flop
   END_IF;
   IF #LINK.Status.ACK OR #FPCMD_RESET_TMR.Q THEN #LINK.Command.RES := FALSE; END_IF;
END_REGION

REGION Network 32: Update Boolean Data in MSW - Bit 16-19: Mode
   // 0 = Auto
   // 1= Single Start
   // 2 = Manual
   // 3= Local
   // 4= Test Mode
   #MSW.EXT.ModeBit1 := #Aoff;
   #MSW.EXT.ModeBit2 := #Aoff;
   #MSW.EXT.ModeBit3 := #Aoff;
   #MSW.EXT.BIT19 := #Aoff;
END_REGION

REGION Network 33: Update Boolean Data in MSW - Bit 21: Alarm Suppressed
   #MSW.EXT.AlarmSuppressed := #ALARM_SupressionActive AND NOT #ALARM_FailureAckRequired;
END_REGION

REGION Network 34: Update Boolean Data in MSW - Bit: 22 Alarm Condition Present
   #MSW.EXT.AlarmPresent := #ALARM_AlarmPresent;
END_REGION

REGION Network 35: Update Boolean Data in MSW - Bit 23: Alarm Failure Present or Unacknowledged
   #MSW.EXT.AlarmFailUnAck := (#AlarmNo >= 1) OR #ALARM_FailureAckRequired;
END_REGION

REGION Network 36: Update Boolean Data in MSW - Bit 24: Alarm Warning Present Or Unacknowledged
   #MSW.EXT.AlarmWarnUnAck := #Aoff;
END_REGION

REGION Network 37: Update Boolean Data in MSW - Bit 25: Acknowledge Required
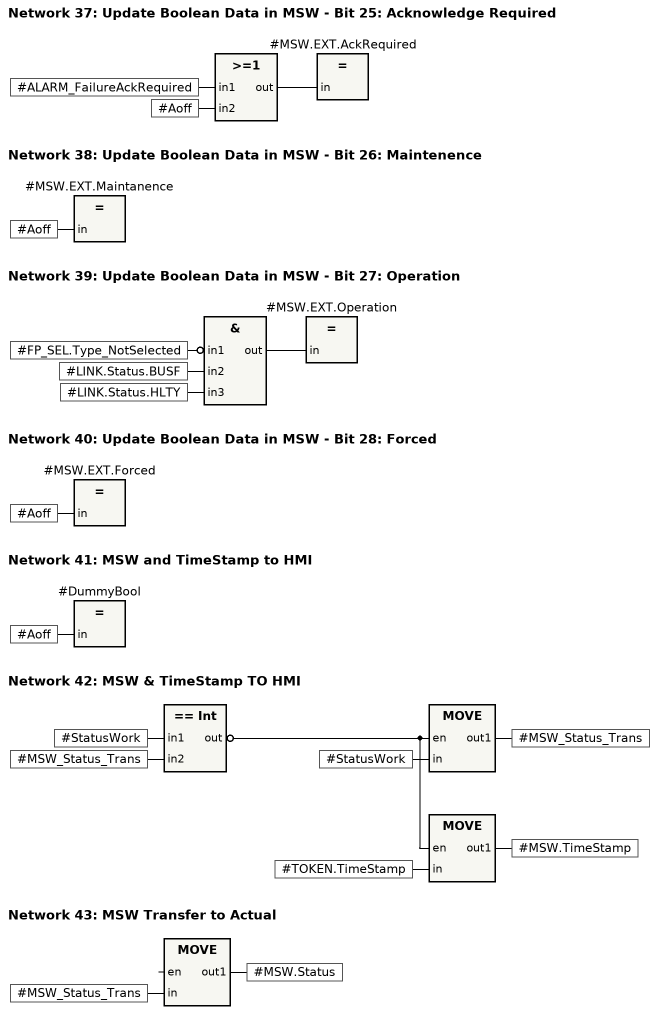
   #MSW.EXT.AckRequired := #ALARM_FailureAckRequired OR #Aoff;
END_REGION

REGION Network 38: Update Boolean Data in MSW - Bit 26: Maintenence
   #MSW.EXT.Maintanence := #Aoff;
END_REGION

REGION Network 39: Update Boolean Data in MSW - Bit 27: Operation
   #MSW.EXT.Operation := NOT #FP_SEL.Type_NotSelected AND #LINK.Status.BUSF AND #LINK.Status.HLTY;
END_REGION

REGION Network 40: Update Boolean Data in MSW - Bit 28: Forced
   #MSW.EXT.Forced := #Aoff;
END_REGION

REGION Network 41: MSW and TimeStamp to HMI
   Done:
   #DummyBool := #Aoff;
END_REGION

REGION Network 42: MSW & TimeStamp TO HMI
   #_w1 := NOT (#StatusWork = #MSW_Status_Trans);
   IF #_w1 THEN
       #MSW_Status_Trans := #StatusWork;
       #MSW.TimeStamp := #TOKEN.TimeStamp;
   END_IF;
END_REGION

REGION Network 43: MSW Transfer to Actual
   #MSW.Status := #MSW_Status_Trans;
END_REGION

REGION Network 44: Token Data to ADAPT
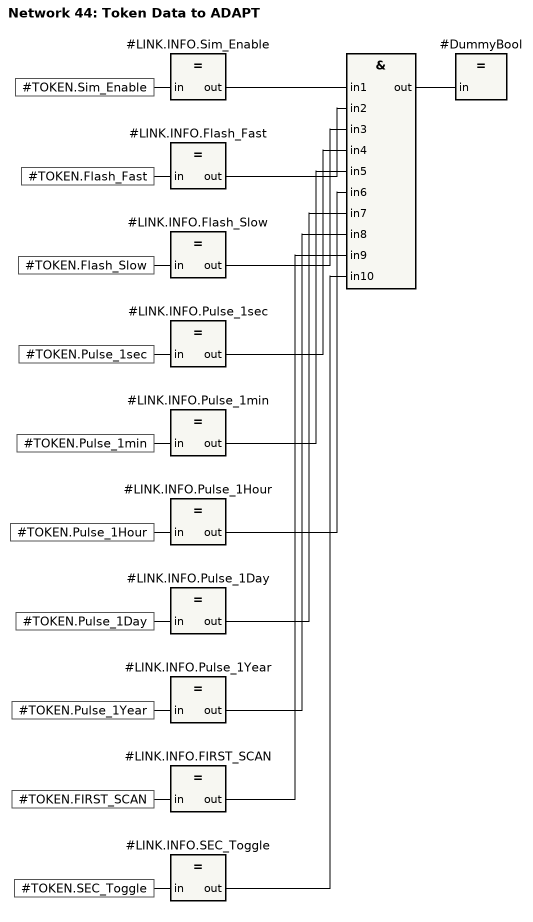
   #LINK.INFO.Sim_Enable := #TOKEN.Sim_Enable;
   #LINK.INFO.Flash_Fast := #TOKEN.Flash_Fast;
   #LINK.INFO.Flash_Slow := #TOKEN.Flash_Slow;
   #LINK.INFO.Pulse_1sec := #TOKEN.Pulse_1sec;
   #LINK.INFO.Pulse_1min := #TOKEN.Pulse_1min;
   #LINK.INFO.Pulse_1Hour := #TOKEN.Pulse_1Hour;
   #LINK.INFO.Pulse_1Day := #TOKEN.Pulse_1Day;
   #LINK.INFO.Pulse_1Year := #TOKEN.Pulse_1Year;
   #LINK.INFO.FIRST_SCAN := #TOKEN.FIRST_SCAN;
   #LINK.INFO.SEC_Toggle := #TOKEN.SEC_Toggle;
   #DummyBool := #TOKEN.Sim_Enable AND #TOKEN.Flash_Fast AND #TOKEN.Flash_Slow AND #TOKEN.Pulse_1sec AND #TOKEN.Pulse_1min AND #TOKEN.Pulse_1Hour AND #TOKEN.Pulse_1Day AND #TOKEN.Pulse_1Year AND #TOKEN.FIRST_SCAN AND #TOKEN.SEC_Toggle;
END_REGION
END_FUNCTION_BLOCK

FUNCTION_BLOCK "ACESYS_LOCATION"   // FB238, FBD
TITLE = ACESYS V8.0 - Build 001 - Location Control
{ S7_Optimized_Access := 'FALSE' }
AUTHOR : Flsmidth
FAMILY : ACESYS
NAME : LOCATION
VERSION : 8.0
   VAR_INPUT
      Master_Link : "ACESYS_MASTER_LINK";
      PLC_CTRL : Bool;   // PLC-based Location Control
      MCS_PERM : Bool;   // Permission to Proximity Location
      PROX : Bool;   // Proximity Tag ID
      CCR_REL : Bool;   // Release Control
      CCR_FR : Bool;   // Force Control
   END_VAR
   VAR_OUTPUT
      MCS : Bool;   // Proximity Location in Control
      MSW : "ACESYS_HMI_STAT_32T";
   END_VAR
   VAR
      OneShot1 : Bool;
      OneShot2 : Bool;
      OneShot3 : Bool;
      OneShot4 : Bool;
      REL_Ons : Bool;
      FR_Ons : Bool;
      Pulse_CCR : Bool;
      Pulse_MCS : Bool;
      TT_CCR : Bool;   // Switch Off Proximity
      TT_MCS : Bool;   // Switch On Proximity
      DummyInt1 : Int;
      DummyInt2 : Int;
      ECSStatusBuilder : Int;
      MSW_Status : Int;
      StatusWork : Int;
      OUT : Struct
         MCS : Bool;
      END_STRUCT;
      MSW_Status_Trans : Int;
   END_VAR
   VAR_TEMP
      Aon : Bool;
      Aoff : Bool;
      DummyBool : Bool;
   END_VAR
   VAR_TEMP   // added for the SCL form of the ladder/FBD networks
      _w1 : Bool;
   END_VAR
BEGIN

REGION Network 1: Always ON
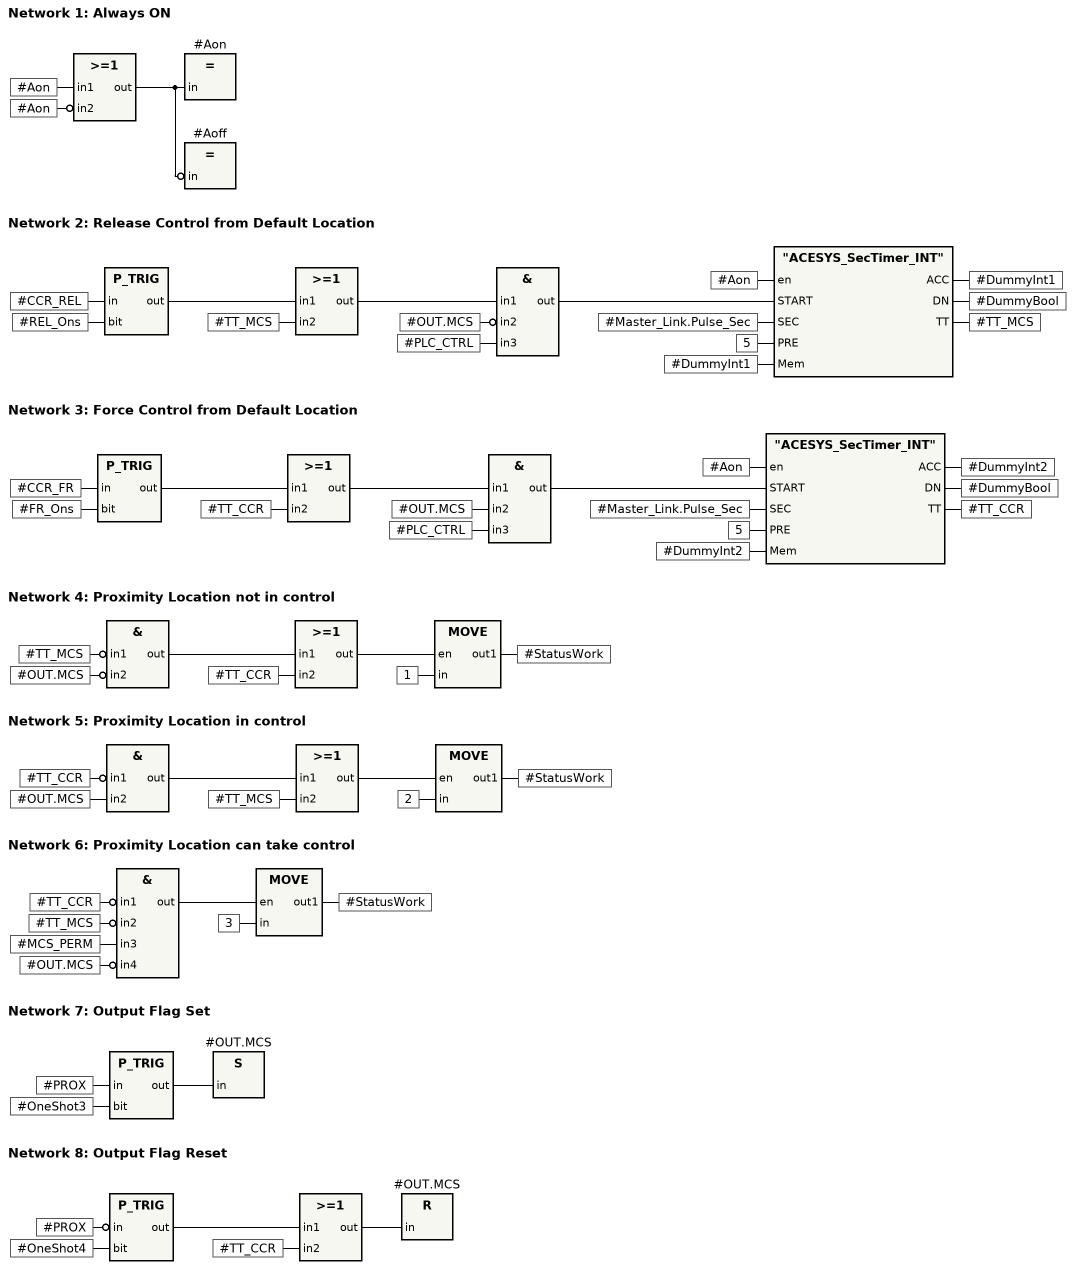
   #Aon := #Aon OR NOT #Aon;
   #Aoff := NOT #Aon;
END_REGION

REGION Network 2: Release Control from Default Location
   #_w1 := #CCR_REL AND NOT #REL_Ons;   // rising edge
   #REL_Ons := #CCR_REL;
   IF #Aon THEN
       "ACESYS_SecTimer_INT"(START := (#_w1 OR #TT_MCS) AND NOT #OUT.MCS AND #PLC_CTRL,
                             SEC := #Master_Link.Pulse_Sec,
                             PRE := 5,
                             Mem := #DummyInt1,
                             ACC => #DummyInt1,
                             DN => #DummyBool,
                             TT => #TT_MCS);
   END_IF;
END_REGION

REGION Network 3: Force Control from Default Location
   #_w1 := #CCR_FR AND NOT #FR_Ons;   // rising edge
   #FR_Ons := #CCR_FR;
   IF #Aon THEN
       "ACESYS_SecTimer_INT"(START := (#_w1 OR #TT_CCR) AND #OUT.MCS AND #PLC_CTRL,
                             SEC := #Master_Link.Pulse_Sec,
                             PRE := 5,
                             Mem := #DummyInt2,
                             ACC => #DummyInt2,
                             DN => #DummyBool,
                             TT => #TT_CCR);
   END_IF;
END_REGION

REGION Network 4: Proximity Location not in control
   IF (NOT #TT_MCS AND NOT #OUT.MCS) OR #TT_CCR THEN #StatusWork := 1; END_IF;
END_REGION

REGION Network 5: Proximity Location in control
   IF (NOT #TT_CCR AND #OUT.MCS) OR #TT_MCS THEN #StatusWork := 2; END_IF;
END_REGION

REGION Network 6: Proximity Location can take control
   IF NOT #TT_CCR AND NOT #TT_MCS AND #MCS_PERM AND NOT #OUT.MCS THEN #StatusWork := 3; END_IF;
END_REGION

REGION Network 7: Output Flag Set
   #_w1 := #PROX AND NOT #OneShot3;   // rising edge
   #OneShot3 := #PROX;
   IF #_w1 THEN #OUT.MCS := TRUE; END_IF;
END_REGION

REGION Network 8: Output Flag Reset
   #_w1 := NOT #PROX AND NOT #OneShot4;   // rising edge
   #OneShot4 := NOT #PROX;
   IF #_w1 OR #TT_CCR THEN #OUT.MCS := FALSE; END_IF;
END_REGION

REGION Network 9: HMI-Based Location Control (V8 to V8 HMI's)
   // Bit 15 = -32768 (HMI-based Location Control)
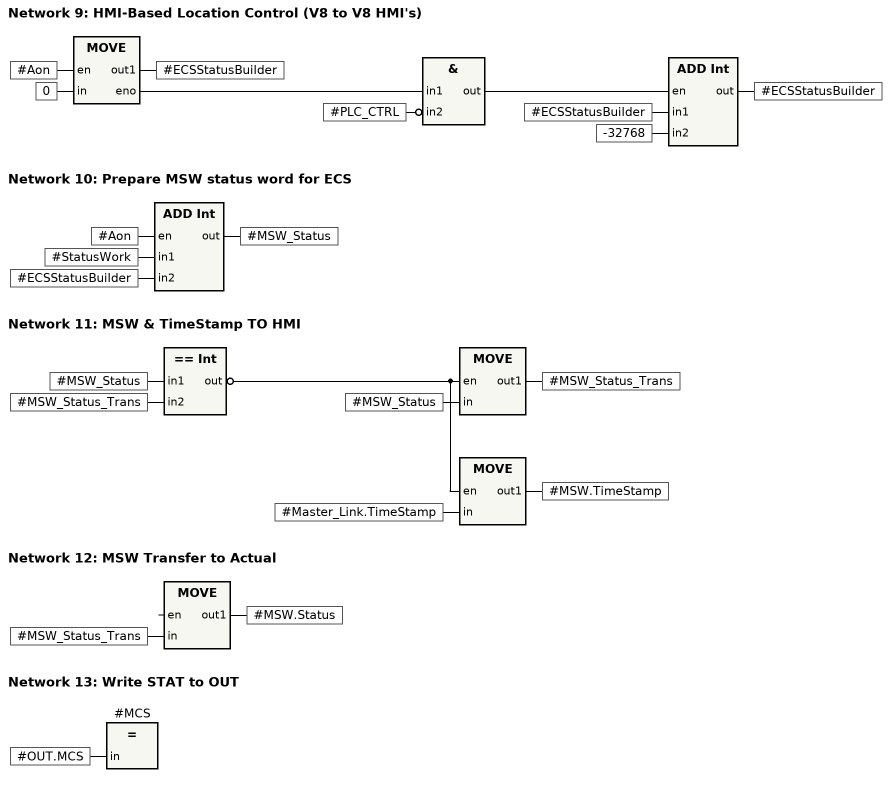
   // ENO of a box is taken as its EN; it also drops when the box reports an error
   IF #Aon THEN #ECSStatusBuilder := 0; END_IF;
   IF #Aon AND NOT #PLC_CTRL THEN #ECSStatusBuilder := #ECSStatusBuilder + (-32768); END_IF;
END_REGION

REGION Network 10: Prepare MSW status word for ECS
   IF #Aon THEN #MSW_Status := #StatusWork + #ECSStatusBuilder; END_IF;
END_REGION

REGION Network 11: MSW & TimeStamp TO HMI
   #_w1 := NOT (#MSW_Status = #MSW_Status_Trans);
   IF #_w1 THEN
       #MSW_Status_Trans := #MSW_Status;
       #MSW.TimeStamp := #Master_Link.TimeStamp;
   END_IF;
END_REGION

REGION Network 12: MSW Transfer to Actual
   #MSW.Status := #MSW_Status_Trans;
END_REGION

REGION Network 13: Write STAT to OUT
   #MCS := #OUT.MCS;
END_REGION
END_FUNCTION_BLOCK

FUNCTION_BLOCK "ACESYS_BQ16_CTRL"   // FB239, FBD
TITLE = ACESYS V8.0 - Build 003 - Air Blaster Control Block
{ S7_Optimized_Access := 'FALSE' }
AUTHOR : FLSmidth
FAMILY : ACESYS
NAME : Air_Ctrl
VERSION : 8.0
// This block is the controlblock for one or more ACESYS_BQ16_PROG
// The block can select and start one program and do manual blast from FP or input 
// pins.
// Data to the programblock(s) shall be send in a datastructure, BQ16_Link, 
// (UDT224)
   VAR_INPUT
      CMD : "ACESYS_GRP_CMD";   // Command
      Config_En : Bool;   // Enable Configuration from Faceplate
      SEL : Bool;   // Unit Select by User Program
      MCS : Bool;   // Local Permission
      LSTR_BQ01 : Bool;   // Local Blast Command
      LSTR_BQ02 : Bool;   // Local Blast Command
      LSTR_BQ03 : Bool;   // Local Blast Command
      LSTR_BQ04 : Bool;   // Local Blast Command
      LSTR_BQ05 : Bool;   // Local Blast Command
      LSTR_BQ06 : Bool;   // Local Blast Command
      LSTR_BQ07 : Bool;   // Local Blast Command
      LSTR_BQ08 : Bool;   // Local Blast Command
      LSTR_BQ09 : Bool;   // Local Blast Command
      LSTR_BQ10 : Bool;   // Local Blast Command
      LSTR_BQ11 : Bool;   // Local Blast Command
      LSTR_BQ12 : Bool;   // Local Blast Command
      LSTR_BQ13 : Bool;   // Local Blast Command
      LSTR_BQ14 : Bool;   // Local Blast Command
      LSTR_BQ15 : Bool;   // Local Blast Command
      LSTR_BQ16 : Bool;   // Local Blast Command
      EXT_MegaBlast : Bool;   // Invoke mega blast
      EXT_ProgCMD : Bool;   // Force Program Command, (Pulse)
      EXT_ProgNO : Int;   // Force Program Number
   END_VAR
   VAR_OUTPUT
      INTL : "ACESYS_INTL";   // Interlock
      INTL_SEQ_STR : "ACESYS_INTL";
      INTL_SEQ_STP : "ACESYS_INTL";
      RUN : Bool;   // Unit Running
      OK : Bool;   // Unit OK
      BQ01_CMD : Bool;   // Blast Command
      BQ02_CMD : Bool;   // Blast Command
      BQ03_CMD : Bool;   // Blast Command
      BQ04_CMD : Bool;   // Blast Command
      BQ05_CMD : Bool;   // Blast Command
      BQ06_CMD : Bool;   // Blast Command
      BQ07_CMD : Bool;   // Blast Command
      BQ08_CMD : Bool;   // Blast Command
      BQ09_CMD : Bool;   // Blast Command
      BQ10_CMD : Bool;   // Blast Command
      BQ11_CMD : Bool;   // Blast Command
      BQ12_CMD : Bool;   // Blast Command
      BQ13_CMD : Bool;   // Blast Command
      BQ14_CMD : Bool;   // Blast Command
      BQ15_CMD : Bool;   // Blast Command
      BQ16_CMD : Bool;   // Blast Command
      ProgAct : Int;   // Active prog. number
      ProgLink : "ACESYS_BQ16";
      MSW : "ACESYS_HMI_STAT_32T";
   END_VAR
   VAR_IN_OUT
      TOKEN : "ACESYS_TOKEN";
   END_VAR
   VAR
      Temp : Int;
      BlockInfo : Struct
         ACESYS_Version : Int;   // Version number
         ACESYS_Build : Int;   // Build Number
         DB_Number : Int;
      END_STRUCT;
      FP_CMD : Struct   // Faceplate Commands
         Man_BQ01 : Bool;   // FacePlateCmd (bit 24): Manual Blast Command
         Man_BQ02 : Bool;   // FacePlateCmd (bit 25): Manual Blast Command
         Man_BQ03 : Bool;   // FacePlateCmd (bit 26): Manual Blast Command
         Man_BQ04 : Bool;   // FacePlateCmd (bit 27): Manual Blast Command
         Man_BQ05 : Bool;   // FacePlateCmd (bit 28): Manual Blast Command
         Man_BQ06 : Bool;   // FacePlateCmd (bit 29): Manual Blast Command
         Man_BQ07 : Bool;   // FacePlateCmd (bit 30): Manual Blast Command
         Man_BQ08 : Bool;   // FacePlateCmd (bit 31): Manual Blast Command
         Man_BQ09 : Bool;   // FacePlateCmd (bit 16): Manual Blast Command
         Man_BQ10 : Bool;   // FacePlateCmd (bit 17): Manual Blast Command
         Man_BQ11 : Bool;   // FacePlateCmd (bit 18): Manual Blast Command
         Man_BQ12 : Bool;   // FacePlateCmd (bit 19): Manual Blast Command
         Man_BQ13 : Bool;   // FacePlateCmd (bit 20): Manual Blast Command
         Man_BQ14 : Bool;   // FacePlateCmd (bit 21): Manual Blast Command
         Man_BQ15 : Bool;   // FacePlateCmd (bit 22): Manual Blast Command
         Man_BQ16 : Bool;   // FacePlateCmd (bit 23): Manual Blast Command
         Start : Bool;   // FacePlateCmd (bit 8): Start Command
         Stop : Bool;   // FacePlateCmd (bit 9): Stop Command
         MegaBlast : Bool;   // FacePlateCmd (bit 10): MegaBlast Command
         QuickStop : Bool;   // FacePlateCmd (bit 11): Quick Stop Command
         w2_Bit12 : Bool;   // FacePlateCmd (bit 12): Spare
         w2_Bit13 : Bool;   // FacePlateCmd (bit 13): Spare
         w2_Bit14 : Bool;   // FacePlateCmd (bit 14): Spare
         Acknowledge : Bool;   // FacePlateCmd (bit 15): ECS Acknowledge
         w2_Bit0 : Bool;   // FacePlateCmd (bit 0): Spare
         w2_Bit1 : Bool;   // FacePlateCmd (bit 1): Spare
         w2_Bit2 : Bool;   // FacePlateCmd (bit 2): Spare
         w2_Bit3 : Bool;   // FacePlateCmd (bit 3): Spare
         w2_Bit4 : Bool;   // FacePlateCmd (bit 4): Spare
         w2_Bit5 : Bool;   // FacePlateCmd (bit 5): Spare
         w2_Bit6 : Bool;   // FacePlateCmd (bit 6): Spare
         w2_Bit7 : Bool;   // FacePlateCmd (bit 7): Spare
      END_STRUCT;
      FP_SEL : Struct   // Faceplate Selections
         Reset : Bool;   // Reset After Stop
         BQ01_Mega : Bool;   // Selected for MegaBlast
         BQ02_Mega : Bool;   // Selected for MegaBlast
         BQ03_Mega : Bool;   // Selected for MegaBlast
         BQ04_Mega : Bool;   // Selected for MegaBlast
         BQ05_Mega : Bool;   // Selected for MegaBlast
         BQ06_Mega : Bool;   // Selected for MegaBlast
         BQ07_Mega : Bool;   // Selected for MegaBlast
         BQ08_Mega : Bool;   // Selected for MegaBlast
         BQ09_Mega : Bool;   // Selected for MegaBlast
         BQ10_Mega : Bool;   // Selected for MegaBlast
         BQ11_Mega : Bool;   // Selected for MegaBlast
         BQ12_Mega : Bool;   // Selected for MegaBlast
         BQ13_Mega : Bool;   // Selected for MegaBlast
         BQ14_Mega : Bool;   // Selected for MegaBlast
         BQ15_Mega : Bool;   // Selected for MegaBlast
         BQ16_Mega : Bool;   // Selected for MegaBlast
         ParentCollection : Bool := TRUE;   // Enable Parent Collection Status
         OutOfService : Bool;   // Select Out of Service
         Spare_Bool_01 : Bool;
         Spare_Bool_02 : Bool;
         Spare_Bool_03 : Bool;
         Spare_Bool_04 : Bool;
         Spare_Bool_05 : Bool;
         Spare_Bool_06 : Bool;
         Spare_Bool_07 : Bool;
         Spare_Bool_08 : Bool;
         Spare_Bool_09 : Bool;
         Spare_Bool_10 : Bool;
         Spare_Bool_11 : Bool;
         Spare_Bool_12 : Bool;
         Spare_Bool_13 : Bool;
      END_STRUCT;
      FP_EN : Struct   // Faceplate Enable Buttons
         PB_QStop : Bool;
         PB_MegaBlast : Bool;
         Mode_SS_FP : Bool := TRUE;
         Spare_Bool_01 : Bool;
         Spare_Bool_02 : Bool;
         Spare_Bool_03 : Bool;
         Spare_Bool_04 : Bool;
         Spare_Bool_05 : Bool;
         Spare_Bool_07 : Bool;
         Spare_Bool_08 : Bool;
         Spare_Bool_09 : Bool;
         Spare_Bool_10 : Bool;
         Spare_Bool_11 : Bool;
         Spare_Bool_12 : Bool;
         Spare_Bool_13 : Bool;
         Spare_Bool_14 : Bool;
      END_STRUCT;
      FP_DIM : Struct   // Faceplate Dimmed Buttons
         Start : Bool;   // 0=DimOut
         Stop : Bool;   // 0=DimOut
         Reset : Bool;   // 0=DimOut
         Force : Bool;   // 0=DimOut (shared by all blasters)
         MegaBlast : Bool;   // 0=DimOut
         QStop : Bool;   // 0=DimOut
         Spare_Bool_01 : Bool;
         Spare_Bool_02 : Bool;
         Spare_Bool_03 : Bool;
         Spare_Bool_04 : Bool;
         Spare_Bool_05 : Bool;
         Spare_Bool_06 : Bool;
         Spare_Bool_07 : Bool;
         Spare_Bool_08 : Bool;
         Spare_Bool_09 : Bool;
         Spare_Bool_10 : Bool;
      END_STRUCT;
      FP_SHOW : Struct   // Faceplate Show Buttons
         PB_Start : Bool;
         PB_Stop : Bool;
         PB_MegaBlast : Bool;
         PB_QStop : Bool;
         Spare_Bool_01 : Bool;
         Spare_Bool_02 : Bool;
         Spare_Bool_03 : Bool;
         Spare_Bool_04 : Bool;
         Spare_Bool_05 : Bool;
         Spare_Bool_06 : Bool;
         Spare_Bool_07 : Bool;
         Spare_Bool_08 : Bool;
         Spare_Bool_09 : Bool;
         Spare_Bool_10 : Bool;
         Spare_Bool_11 : Bool;
         Spare_Bool_12 : Bool;
      END_STRUCT;
      FP_PARM : Struct   // Faceplate Parameters
         NoOfBlasters : Int := 16;   // Number of Blasters to be Used
         Spare_Int_01 : Int;
         Prog_SP : Int;   // Program SP from FP
         NoProgram_PV : Int;   // Number of Programs, PV
         ForceTime_SP : Int := 1000;   // Force Time SP from FP
         MegaBlastTime_SP : Int := 1000;   // MegaBlast Time SP from FP
         StopReason : Int;
         INTL : Bool;   // Interlock
         INTL_SEQ_STR1 : Bool;   // Interlock Sequence Start
         INTL_SEQ_STP : Bool;   // Interlock Sequence Stop
         ASTR : Bool;   // Auto Start
         SACK : Bool;   // SACK
         Spare_Bool_03 : Bool;
         Spare_Bool_04 : Bool;
         Spare_Bool_05 : Bool;
         Spare_Bool_06 : Bool;
         Spare_Bool_07 : Bool;
         Spare_Bool_08 : Bool;
         Spare_Bool_09 : Bool;
         Spare_Bool_10 : Bool;
         Spare_Bool_11 : Bool;
         Spare_Bool_12 : Bool;
         Spare_Bool_13 : Bool;
         BQ01_CNT : DInt;   // Blast Counter
         BQ02_CNT : DInt;   // Blast Counter
         BQ03_CNT : DInt;   // Blast Counter
         BQ04_CNT : DInt;   // Blast Counter
         BQ05_CNT : DInt;   // Blast Counter
         BQ06_CNT : DInt;   // Blast Counter
         BQ07_CNT : DInt;   // Blast Counter
         BQ08_CNT : DInt;   // Blast Counter
         BQ09_CNT : DInt;   // Blast Counter
         BQ10_CNT : DInt;   // Blast Counter
         BQ11_CNT : DInt;   // Blast Counter
         BQ12_CNT : DInt;   // Blast Counter
         BQ13_CNT : DInt;   // Blast Counter
         BQ14_CNT : DInt;   // Blast Counter
         BQ15_CNT : DInt;   // Blast Counter
         BQ16_CNT : DInt;   // Blast Counter
         BQ01_CMD_IND : Bool;   // FP Delayed CMD Indication
         BQ02_CMD_IND : Bool;   // FP Delayed CMD Indication
         BQ03_CMD_IND : Bool;   // FP Delayed CMD Indication
         BQ04_CMD_IND : Bool;   // FP Delayed CMD Indication
         BQ05_CMD_IND : Bool;   // FP Delayed CMD Indication
         BQ06_CMD_IND : Bool;   // FP Delayed CMD Indication
         BQ07_CMD_IND : Bool;   // FP Delayed CMD Indication
         BQ08_CMD_IND : Bool;   // FP Delayed CMD Indication
         BQ09_CMD_IND : Bool;   // FP Delayed CMD Indication
         BQ10_CMD_IND : Bool;   // FP Delayed CMD Indication
         BQ11_CMD_IND : Bool;   // FP Delayed CMD Indication
         BQ12_CMD_IND : Bool;   // FP Delayed CMD Indication
         BQ13_CMD_IND : Bool;   // FP Delayed CMD Indication
         BQ14_CMD_IND : Bool;   // FP Delayed CMD Indication
         BQ15_CMD_IND : Bool;   // FP Delayed CMD Indication
         BQ16_CMD_IND : Bool;   // FP Delayed CMD Indication
         BQ01_CNT_RST : Bool;   // Reset Blast Counter
         BQ02_CNT_RST : Bool;   // Reset Blast Counter
         BQ03_CNT_RST : Bool;   // Reset Blast Counter
         BQ04_CNT_RST : Bool;   // Reset Blast Counter
         BQ05_CNT_RST : Bool;   // Reset Blast Counter
         BQ06_CNT_RST : Bool;   // Reset Blast Counter
         BQ07_CNT_RST : Bool;   // Reset Blast Counter
         BQ08_CNT_RST : Bool;   // Reset Blast Counter
         BQ09_CNT_RST : Bool;   // Reset Blast Counter
         BQ10_CNT_RST : Bool;   // Reset Blast Counter
         BQ11_CNT_RST : Bool;   // Reset Blast Counter
         BQ12_CNT_RST : Bool;   // Reset Blast Counter
         BQ13_CNT_RST : Bool;   // Reset Blast Counter
         BQ14_CNT_RST : Bool;   // Reset Blast Counter
         BQ15_CNT_RST : Bool;   // Reset Blast Counter
         BQ16_CNT_RST : Bool;   // Reset Blast Counter
      END_STRUCT;
      ForceTime : Time;
      MegaBlastTime : Time;
      Old_Prog_SP : Int;   // Old Program SP
      StatusWork : Int;   // MSW Status
      MSW_Status : Int;
      Select : Bool;   // Group & Unit Selected
      Spare_Bool_01 : Bool;
      Spare_Bool_02 : Bool;
      Spare_Bool_03 : Bool;
      Spare_Bool_04 : Bool;
      Spare_Bool_05 : Bool;
      Spare_Bool_06 : Bool;
      Spare_Bool_07 : Bool;
      Spare_Bool_08 : Bool;
      Spare_Bool_09 : Bool;
      Spare_Bool_10 : Bool;
      Spare_Bool_11 : Bool;
      Spare_Bool_12 : Bool;
      Spare_Bool_13 : Bool;
      Spare_Bool_14 : Bool;
      Spare_Bool_15 : Bool;
      CMD_Int : Struct
         Start : Bool;   // FP Start Command
         Stop : Bool;   // FP Stop Command
         Reset : Bool;   // FP (1=Reset after Stop)
         Mega : Bool;   // Mega blast requested
         QuickStop : Bool;   // FP Quick Stop Command
         Spare_Bool_01 : Bool;
         Spare_Bool_02 : Bool;
         Spare_Bool_03 : Bool;
         Spare_Bool_04 : Bool;
         Spare_Bool_05 : Bool;
         Spare_Bool_06 : Bool;
         Spare_Bool_07 : Bool;
         Spare_Bool_08 : Bool;
         Spare_Bool_09 : Bool;
         Spare_Bool_10 : Bool;
         Spare_Bool_11 : Bool;
      END_STRUCT;
      STATE : Struct
         Running : Bool;   // State - Unit Running
         Selected : Bool;   // State - Unit Selected
         SelToStop : Bool;   // State - Selected to Stop
         SingleStart : Bool;   // State - Single Start Mode
         Stopped : Bool;   // State - Unit Stopped
         Interlocked : Bool;   // State - Interlocked
         SEQInterlocked : Bool;   // State - Sequence Interlocked
         Aux_SelToStop : Bool;   // One Scan Delay
         AutoStart : Bool;   // State - Auto Start
         Spare_Bool_03 : Bool;
         Spare_Bool_04 : Bool;
         Spare_Bool_05 : Bool;
         Spare_Bool_06 : Bool;
         Spare_Bool_07 : Bool;
         Spare_Bool_08 : Bool;
         Spare_Bool_09 : Bool;
      END_STRUCT;
      TMR : Struct
         BQ01_DN : Bool;   // Timer Done
         BQ02_DN : Bool;   // Timer Done
         BQ03_DN : Bool;   // Timer Done
         BQ04_DN : Bool;   // Timer Done
         BQ05_DN : Bool;   // Timer Done
         BQ06_DN : Bool;   // Timer Done
         BQ07_DN : Bool;   // Timer Done
         BQ08_DN : Bool;   // Timer Done
         BQ09_DN : Bool;   // Timer Done
         BQ10_DN : Bool;   // Timer Done
         BQ11_DN : Bool;   // Timer Done
         BQ12_DN : Bool;   // Timer Done
         BQ13_DN : Bool;   // Timer Done
         BQ14_DN : Bool;   // Timer Done
         BQ15_DN : Bool;   // Timer Done
         BQ16_DN : Bool;   // Timer Done
         BQ01_mem : Int;   // Timer memory
         BQ02_mem : Int;   // Timer memory
         BQ03_mem : Int;   // Timer memory
         BQ04_mem : Int;   // Timer memory
         BQ05_mem : Int;   // Timer memory
         BQ06_mem : Int;   // Timer memory
         BQ07_mem : Int;   // Timer memory
         BQ08_mem : Int;   // Timer memory
         BQ09_mem : Int;   // Timer memory
         BQ10_mem : Int;   // Timer memory
         BQ11_mem : Int;   // Timer memory
         BQ12_mem : Int;   // Timer memory
         BQ13_mem : Int;   // Timer memory
         BQ14_mem : Int;   // Timer memory
         BQ15_mem : Int;   // Timer memory
         BQ16_mem : Int;   // Timer memory
      END_STRUCT;
      ONS : Struct
         Pulse01 : Bool;   // Oneshoot External Program Change
         Pulse02 : Bool;   // Oneshoot Counter
         Pulse03 : Bool;   // Oneshoot Counter
         Pulse04 : Bool;   // Oneshoot Counter
         Pulse05 : Bool;   // Oneshoot Counter
         Pulse06 : Bool;   // Oneshoot Counter
         Pulse07 : Bool;   // Oneshoot Counter
         Pulse08 : Bool;   // Oneshoot Counter
         Pulse09 : Bool;   // Oneshoot Counter
         Pulse10 : Bool;   // Oneshoot Counter
         Pulse11 : Bool;   // Oneshoot Counter
         Pulse12 : Bool;   // Oneshoot Counter
         Pulse13 : Bool;   // Oneshoot Counter
         Pulse14 : Bool;   // Oneshoot Counter
         Pulse15 : Bool;   // Oneshoot Counter
         Pulse16 : Bool;   // Oneshoot Counter
         Pulse17 : Bool;   // Oneshoot Counter
         Pulse20 : Bool;   // Oneshoot Local blast detected
         Pulse21 : Bool;   // Oneshoot Local blast detected
         Pulse22 : Bool;   // Oneshoot Local blast detected
         Pulse23 : Bool;   // Oneshoot Local blast detected
         Pulse24 : Bool;   // Oneshoot Local blast detected
         Pulse25 : Bool;   // Oneshoot Local blast detected
         Pulse26 : Bool;   // Oneshoot Local blast detected
         Pulse27 : Bool;   // Oneshoot Local blast detected
         Pulse28 : Bool;   // Oneshoot Local blast detected
         Pulse29 : Bool;   // Oneshoot Local blast detected
         Pulse30 : Bool;   // Spare
         Pulse31 : Bool;   // Oneshoot Local blast detected
         Pulse32 : Bool;   // Oneshoot Local blast detected
         Pulse33 : Bool;   // Oneshoot Local blast detected
         Pulse34 : Bool;   // Oneshoot Local blast detected
         Pulse35 : Bool;   // Oneshoot Local blast detected
         Pulse36 : Bool;   // Oneshoot Local blast detected
         PulseMega : Bool;   // Oneshoot External MegaBlast
         Spare_Bool_01 : Bool;
         Spare_Bool_02 : Bool;
         Spare_Bool_03 : Bool;
         Spare_Bool_04 : Bool;
         Spare_Bool_05 : Bool;
         Spare_Bool_06 : Bool;
         Spare_Bool_07 : Bool;
         Spare_Bool_08 : Bool;
         Spare_Bool_09 : Bool;
         Spare_Bool_10 : Bool;
         Spare_Bool_11 : Bool;
         Spare_Bool_12 : Bool;
         Spare_Bool_13 : Bool;
      END_STRUCT;
      OUT : Struct
         ProgLink_ProgramIncrement : Int;
         ProgLink_SelectProgram : Int;
         ProgLink_BQ_CMD : Array[0..16] of Bool;
         INTL_OK : Bool;
         INTL_SEQ_STR_OK : Bool;
         INTL_SEQ_STP_OK : Bool;
         RUN : Bool;
         OK : Bool;
         BQ01_CMD : Bool;
         BQ02_CMD : Bool;
         BQ03_CMD : Bool;
         BQ04_CMD : Bool;
         BQ05_CMD : Bool;
         BQ06_CMD : Bool;
         BQ07_CMD : Bool;
         BQ08_CMD : Bool;
         BQ09_CMD : Bool;
         BQ10_CMD : Bool;
         BQ11_CMD : Bool;
         BQ12_CMD : Bool;
         BQ13_CMD : Bool;
         BQ14_CMD : Bool;
         BQ15_CMD : Bool;
         BQ16_CMD : Bool;
      END_STRUCT;
      BQ01_ManBlast : TOF_TIME;
      BQ02_ManBlast : TOF_TIME;
      BQ03_ManBlast : TOF_TIME;
      BQ04_ManBlast : TOF_TIME;
      BQ05_ManBlast : TOF_TIME;
      BQ06_ManBlast : TOF_TIME;
      BQ07_ManBlast : TOF_TIME;
      BQ08_ManBlast : TOF_TIME;
      BQ09_ManBlast : TOF_TIME;
      BQ10_ManBlast : TOF_TIME;
      BQ11_ManBlast : TOF_TIME;
      BQ12_ManBlast : TOF_TIME;
      BQ13_ManBlast : TOF_TIME;
      BQ14_ManBlast : TOF_TIME;
      BQ15_ManBlast : TOF_TIME;
      BQ16_ManBlast : TOF_TIME;
      BlastTimer : TON_TIME;
   END_VAR
   VAR_TEMP
      Aon : Bool;   // Always on
      Aoff : Bool;   // Alway off
      DummyBool : Bool;
      DummyInt : Int;
      DummyDint : DInt;
      Temp_RUN : Bool;
   END_VAR
   VAR_TEMP   // added for the SCL form of the ladder/FBD networks
      _w1 : Bool;
      _w2 : Bool;
      _w3 : Bool;
      _w4 : Bool;
      _w5 : Bool;
      _w6 : Bool;
   END_VAR
BEGIN

REGION Network 1: Aon/Aoff Definition
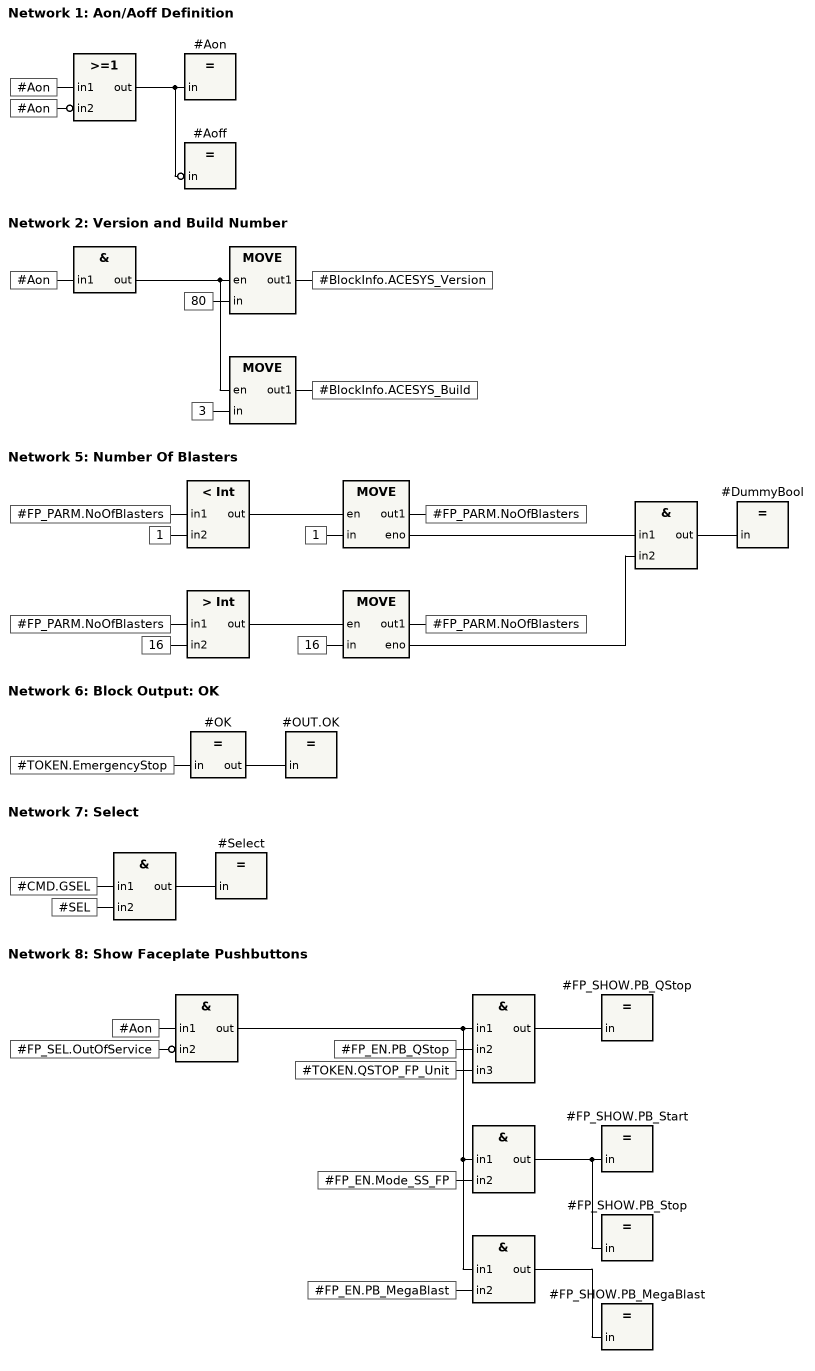
   #Aon := #Aon OR NOT #Aon;
   #Aoff := NOT #Aon;
END_REGION

REGION Network 2: Version and Build Number
   IF #Aon THEN
       #BlockInfo.ACESYS_Version := 80;
       #BlockInfo.ACESYS_Build := 3;
   END_IF;
END_REGION

REGION Network 3 (STL): Instance DB Number to Faceplate
         L     DINO;
         T     #BlockInfo.DB_Number;
END_REGION

REGION Network 4 (SCL): Transfer Current Output Status to Internal Flags (Dependent on DB offsets - update if changed)
   // These outputs can be changed from outside the block, need to acquire their current state
   // Note: Integers are stored with bytes swapped (byte 29: will work as long as programs are less than 255)
   #OUT.INTL_OK := PEEK_BOOL(area := 16#84, dbNumber := #BlockInfo.DB_Number, byteOffset := 8, bitOffset := 0);
   #OUT.INTL_SEQ_STR_OK := PEEK_BOOL(area := 16#84, dbNumber := #BlockInfo.DB_Number, byteOffset := 10, bitOffset := 0);
   #OUT.INTL_SEQ_STP_OK := PEEK_BOOL(area := 16#84, dbNumber := #BlockInfo.DB_Number, byteOffset := 12, bitOffset := 0);
   #OUT.ProgLink_ProgramIncrement := PEEK(area := 16#84, dbNumber := #BlockInfo.DB_Number, byteOffset := 29);
   #OUT.ProgLink_BQ_CMD[1] := PEEK_BOOL(area := 16#84, dbNumber := #BlockInfo.DB_Number, byteOffset := 22, bitOffset := 1);
   #OUT.ProgLink_BQ_CMD[2] := PEEK_BOOL(area := 16#84, dbNumber := #BlockInfo.DB_Number, byteOffset := 22, bitOffset := 2);
   #OUT.ProgLink_BQ_CMD[3] := PEEK_BOOL(area := 16#84, dbNumber := #BlockInfo.DB_Number, byteOffset := 22, bitOffset := 3);
   #OUT.ProgLink_BQ_CMD[4] := PEEK_BOOL(area := 16#84, dbNumber := #BlockInfo.DB_Number, byteOffset := 22, bitOffset := 4);
   #OUT.ProgLink_BQ_CMD[5] := PEEK_BOOL(area := 16#84, dbNumber := #BlockInfo.DB_Number, byteOffset := 22, bitOffset := 5);
   #OUT.ProgLink_BQ_CMD[6] := PEEK_BOOL(area := 16#84, dbNumber := #BlockInfo.DB_Number, byteOffset := 22, bitOffset := 6);
   #OUT.ProgLink_BQ_CMD[7] := PEEK_BOOL(area := 16#84, dbNumber := #BlockInfo.DB_Number, byteOffset := 22, bitOffset := 7);
   #OUT.ProgLink_BQ_CMD[8] := PEEK_BOOL(area := 16#84, dbNumber := #BlockInfo.DB_Number, byteOffset := 23, bitOffset := 0);
   #OUT.ProgLink_BQ_CMD[9] := PEEK_BOOL(area := 16#84, dbNumber := #BlockInfo.DB_Number, byteOffset := 23, bitOffset := 1);
   #OUT.ProgLink_BQ_CMD[10] := PEEK_BOOL(area := 16#84, dbNumber := #BlockInfo.DB_Number, byteOffset := 23, bitOffset := 2);
   #OUT.ProgLink_BQ_CMD[11] := PEEK_BOOL(area := 16#84, dbNumber := #BlockInfo.DB_Number, byteOffset := 23, bitOffset := 3);
   #OUT.ProgLink_BQ_CMD[12] := PEEK_BOOL(area := 16#84, dbNumber := #BlockInfo.DB_Number, byteOffset := 23, bitOffset := 4);
   #OUT.ProgLink_BQ_CMD[13] := PEEK_BOOL(area := 16#84, dbNumber := #BlockInfo.DB_Number, byteOffset := 23, bitOffset := 5);
   #OUT.ProgLink_BQ_CMD[14] := PEEK_BOOL(area := 16#84, dbNumber := #BlockInfo.DB_Number, byteOffset := 23, bitOffset := 6);
   #OUT.ProgLink_BQ_CMD[15] := PEEK_BOOL(area := 16#84, dbNumber := #BlockInfo.DB_Number, byteOffset := 23, bitOffset := 7);
   #OUT.ProgLink_BQ_CMD[16] := PEEK_BOOL(area := 16#84, dbNumber := #BlockInfo.DB_Number, byteOffset := 24, bitOffset := 0);
END_REGION

REGION Network 5: Number Of Blasters
   // Allowed range 1 - 16
   // ENO of a box is taken as its EN; it also drops when the box reports an error
   #_w1 := #FP_PARM.NoOfBlasters < 1;
   IF #_w1 THEN #FP_PARM.NoOfBlasters := 1; END_IF;
   #_w2 := #FP_PARM.NoOfBlasters > 16;
   IF #_w2 THEN #FP_PARM.NoOfBlasters := 16; END_IF;
   #DummyBool := #_w1 AND #_w2;
END_REGION

REGION Network 6: Block Output: OK
   #OK := #TOKEN.EmergencyStop;
   #OUT.OK := #TOKEN.EmergencyStop;
END_REGION

REGION Network 7: Select
   #Select := #CMD.GSEL AND #SEL;
END_REGION

REGION Network 8: Show Faceplate Pushbuttons
   #_w1 := #Aon AND NOT #FP_SEL.OutOfService;
   #FP_SHOW.PB_QStop := #_w1 AND #FP_EN.PB_QStop AND #TOKEN.QSTOP_FP_Unit;
   #FP_SHOW.PB_Start := #_w1 AND #FP_EN.Mode_SS_FP;
   #FP_SHOW.PB_Stop := #FP_SHOW.PB_Start;
   #FP_SHOW.PB_MegaBlast := #_w1 AND #FP_EN.PB_MegaBlast;
END_REGION

REGION Network 9: DimOut Faceplate Pushbuttons
   // Build 003-11 Aug 2021- SURAM-IN- State Running modified with Autostart
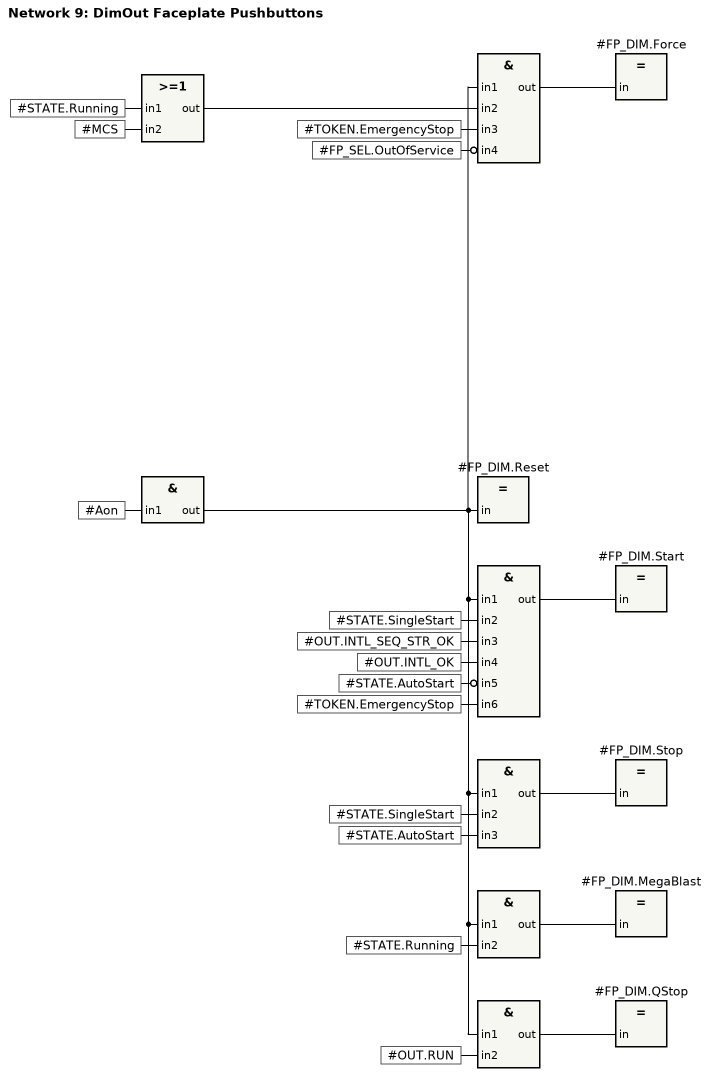
   #FP_DIM.Reset := #Aon;
   #FP_DIM.Force := #Aon AND (#STATE.Running OR #MCS) AND #TOKEN.EmergencyStop AND NOT #FP_SEL.OutOfService;
   #FP_DIM.Start := #Aon AND #STATE.SingleStart AND #OUT.INTL_SEQ_STR_OK AND #OUT.INTL_OK AND NOT #STATE.AutoStart AND #TOKEN.EmergencyStop;
   #FP_DIM.Stop := #Aon AND #STATE.SingleStart AND #STATE.AutoStart;
   #FP_DIM.MegaBlast := #Aon AND #STATE.Running;
   #FP_DIM.QStop := #Aon AND #OUT.RUN;
END_REGION

REGION Network 10: Commands from Faceplate
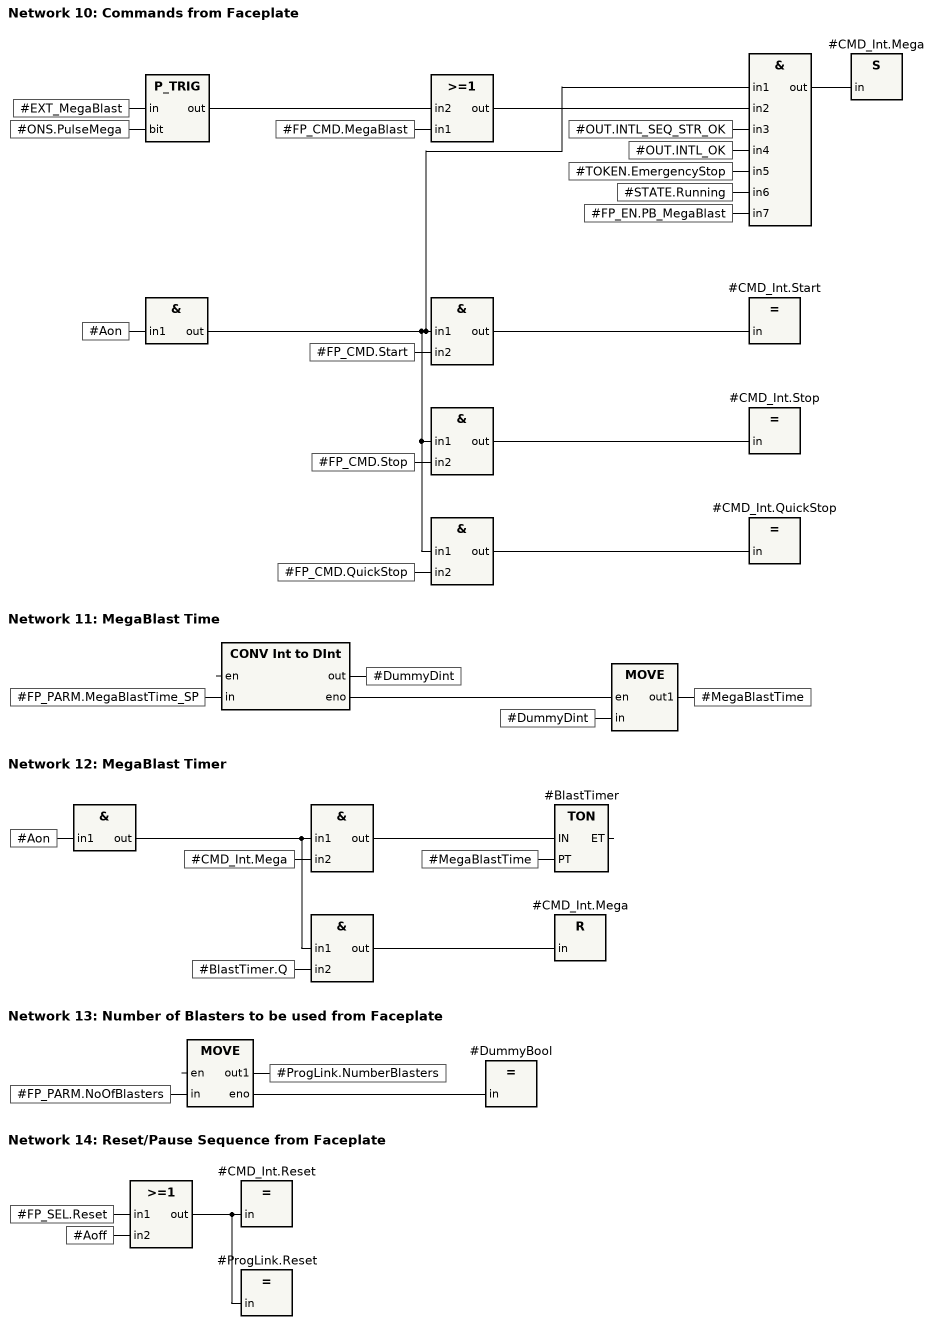
   #CMD_Int.Start := #Aon AND #FP_CMD.Start;
   #CMD_Int.Stop := #Aon AND #FP_CMD.Stop;
   #CMD_Int.QuickStop := #Aon AND #FP_CMD.QuickStop;
   #_w1 := #EXT_MegaBlast AND NOT #ONS.PulseMega;   // rising edge
   #ONS.PulseMega := #EXT_MegaBlast;
   IF #Aon AND (#_w1 OR #FP_CMD.MegaBlast) AND #OUT.INTL_SEQ_STR_OK AND #OUT.INTL_OK AND #TOKEN.EmergencyStop AND #STATE.Running AND #FP_EN.PB_MegaBlast THEN
       #CMD_Int.Mega := TRUE;
   END_IF;
END_REGION

REGION Network 11: MegaBlast Time
   // ENO of a box is taken as its EN; it also drops when the box reports an error
   #DummyDint := INT_TO_DINT(#FP_PARM.MegaBlastTime_SP);
   #MegaBlastTime := #DummyDint;
END_REGION

REGION Network 12: MegaBlast Timer
   #BlastTimer(IN := #Aon AND #CMD_Int.Mega, PT := #MegaBlastTime);   // TON
   IF #Aon AND #BlastTimer.Q THEN #CMD_Int.Mega := FALSE; END_IF;
END_REGION

REGION Network 13: Number of Blasters to be used from Faceplate
   // ENO of a box is taken as its EN; it also drops when the box reports an error
   #ProgLink.NumberBlasters := #FP_PARM.NoOfBlasters;
   #DummyBool := TRUE;
END_REGION

REGION Network 14: Reset/Pause Sequence from Faceplate
   #CMD_Int.Reset := #FP_SEL.Reset OR #Aoff;
   #ProgLink.Reset := #CMD_Int.Reset;
END_REGION

REGION Network 15: Get Total Number of Programs
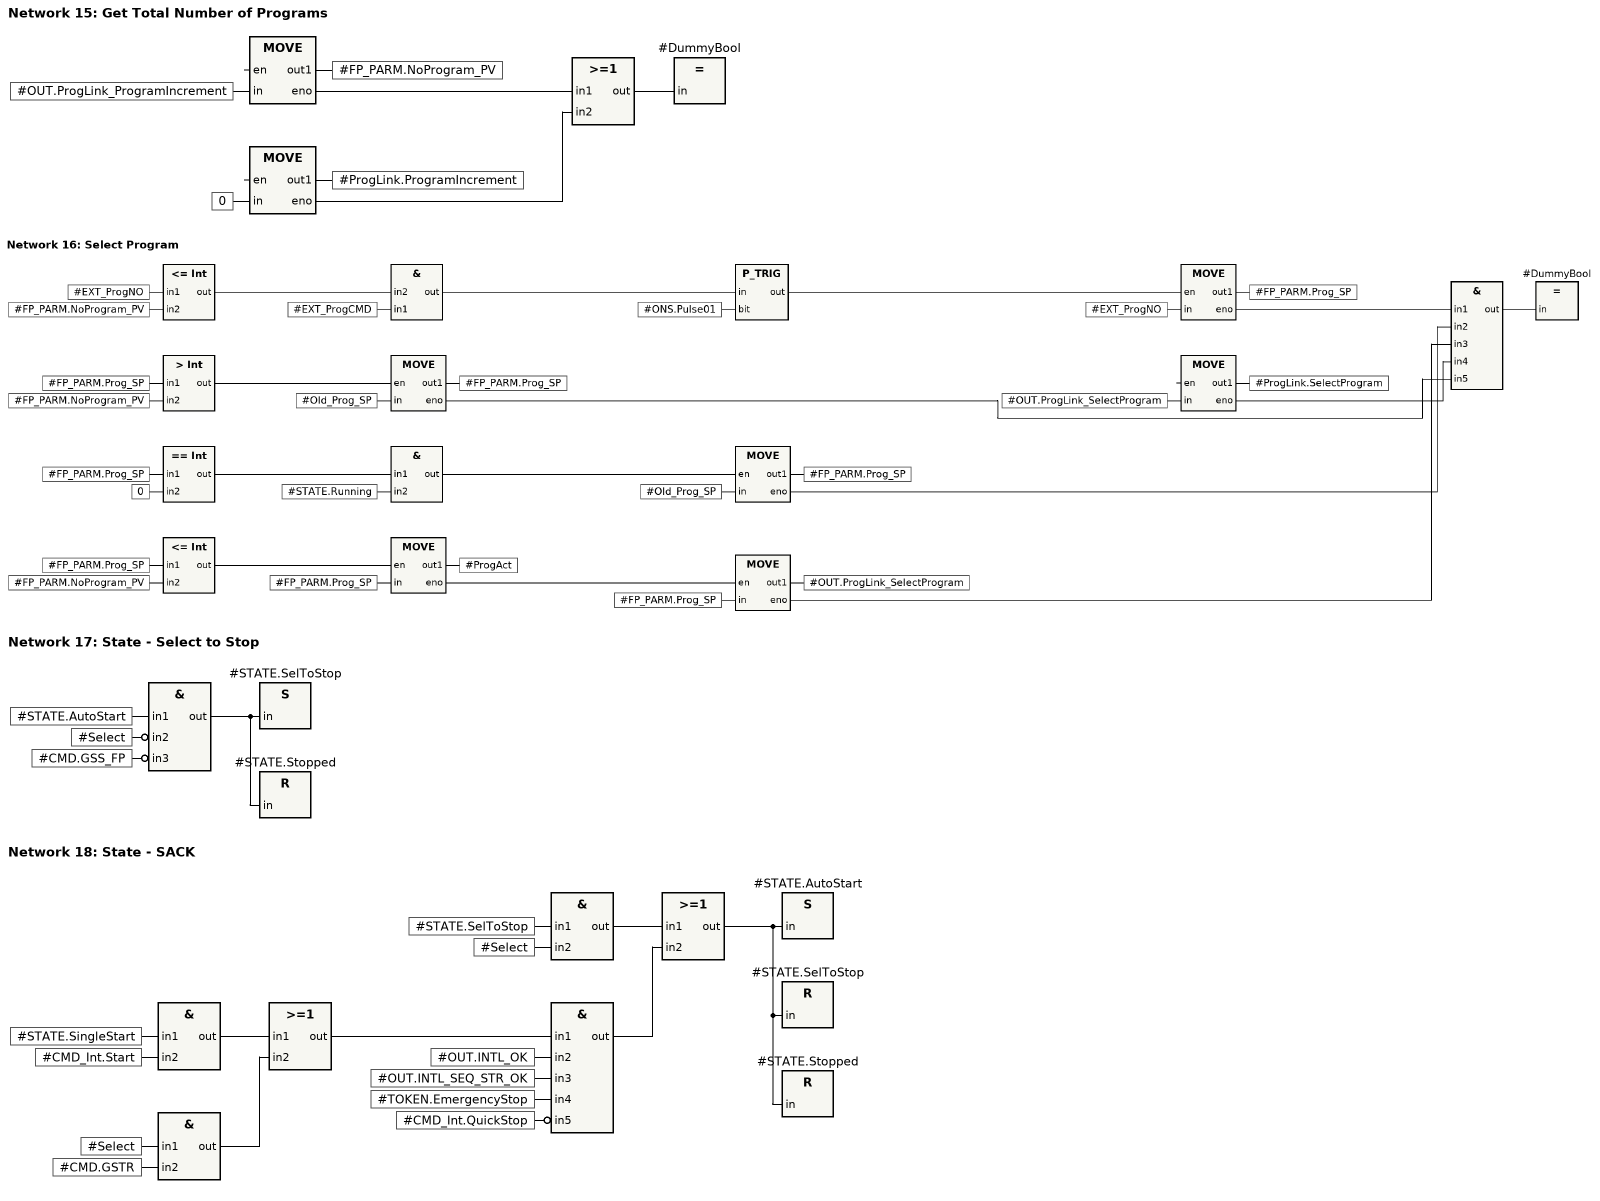
   #FP_PARM.NoProgram_PV := #OUT.ProgLink_ProgramIncrement;
   #ProgLink.ProgramIncrement := 0;
   #DummyBool := TRUE OR TRUE;
END_REGION

REGION Network 16: Select Program
   // From faceplate or from input-pin trigged by a force command (pulse)
   // ENO of a box is taken as its EN; it also drops when the box reports an error
   #_w1 := (#EXT_ProgNO <= #FP_PARM.NoProgram_PV) AND #EXT_ProgCMD;
   #_w2 := #_w1 AND NOT #ONS.Pulse01;   // rising edge
   #ONS.Pulse01 := #_w1;
   IF #_w2 THEN #FP_PARM.Prog_SP := #EXT_ProgNO; END_IF;
   #_w3 := (#FP_PARM.Prog_SP = 0) AND #STATE.Running;
   IF #_w3 THEN #FP_PARM.Prog_SP := #Old_Prog_SP; END_IF;
   #_w4 := #FP_PARM.Prog_SP <= #FP_PARM.NoProgram_PV;
   IF #_w4 THEN
       #ProgAct := #FP_PARM.Prog_SP;
       #OUT.ProgLink_SelectProgram := #FP_PARM.Prog_SP;
   END_IF;
   #ProgLink.SelectProgram := #OUT.ProgLink_SelectProgram;
   #_w5 := #FP_PARM.Prog_SP > #FP_PARM.NoProgram_PV;
   IF #_w5 THEN #FP_PARM.Prog_SP := #Old_Prog_SP; END_IF;
   #DummyBool := #_w2 AND #_w3 AND #_w4 AND #_w5;
END_REGION

REGION Network 17: State - Select to Stop
   // Build 003-11 Aug 2021- SURAM-IN- State Running modified with Autostart
   IF #STATE.AutoStart AND NOT #Select AND NOT #CMD.GSS_FP THEN
       #STATE.SelToStop := TRUE;
       #STATE.Stopped := FALSE;
   END_IF;
END_REGION

REGION Network 18: State - SACK
   // Build 003-11 Aug 2021- SURAM-IN- New State Auto Start Logic Derived
   IF (#STATE.SelToStop AND #Select) OR (((#STATE.SingleStart AND #CMD_Int.Start) OR (#Select AND #CMD.GSTR)) AND #OUT.INTL_OK AND #OUT.INTL_SEQ_STR_OK AND #TOKEN.EmergencyStop AND NOT #CMD_Int.QuickStop) THEN
       #STATE.AutoStart := TRUE;
   END_IF;
   #_w1 := (#STATE.SelToStop AND #Select) OR (((#STATE.SingleStart AND #CMD_Int.Start) OR (#Select AND #CMD.GSTR)) AND #OUT.INTL_OK AND #OUT.INTL_SEQ_STR_OK AND #TOKEN.EmergencyStop AND NOT #CMD_Int.QuickStop);
   IF #_w1 THEN
       #STATE.SelToStop := FALSE;
       #STATE.Stopped := FALSE;
   END_IF;
END_REGION

REGION Network 19: State - Running
   // Build 003-10 Aug 2021- SURAM-IN- State Running Logic modified to support Auto Start Function
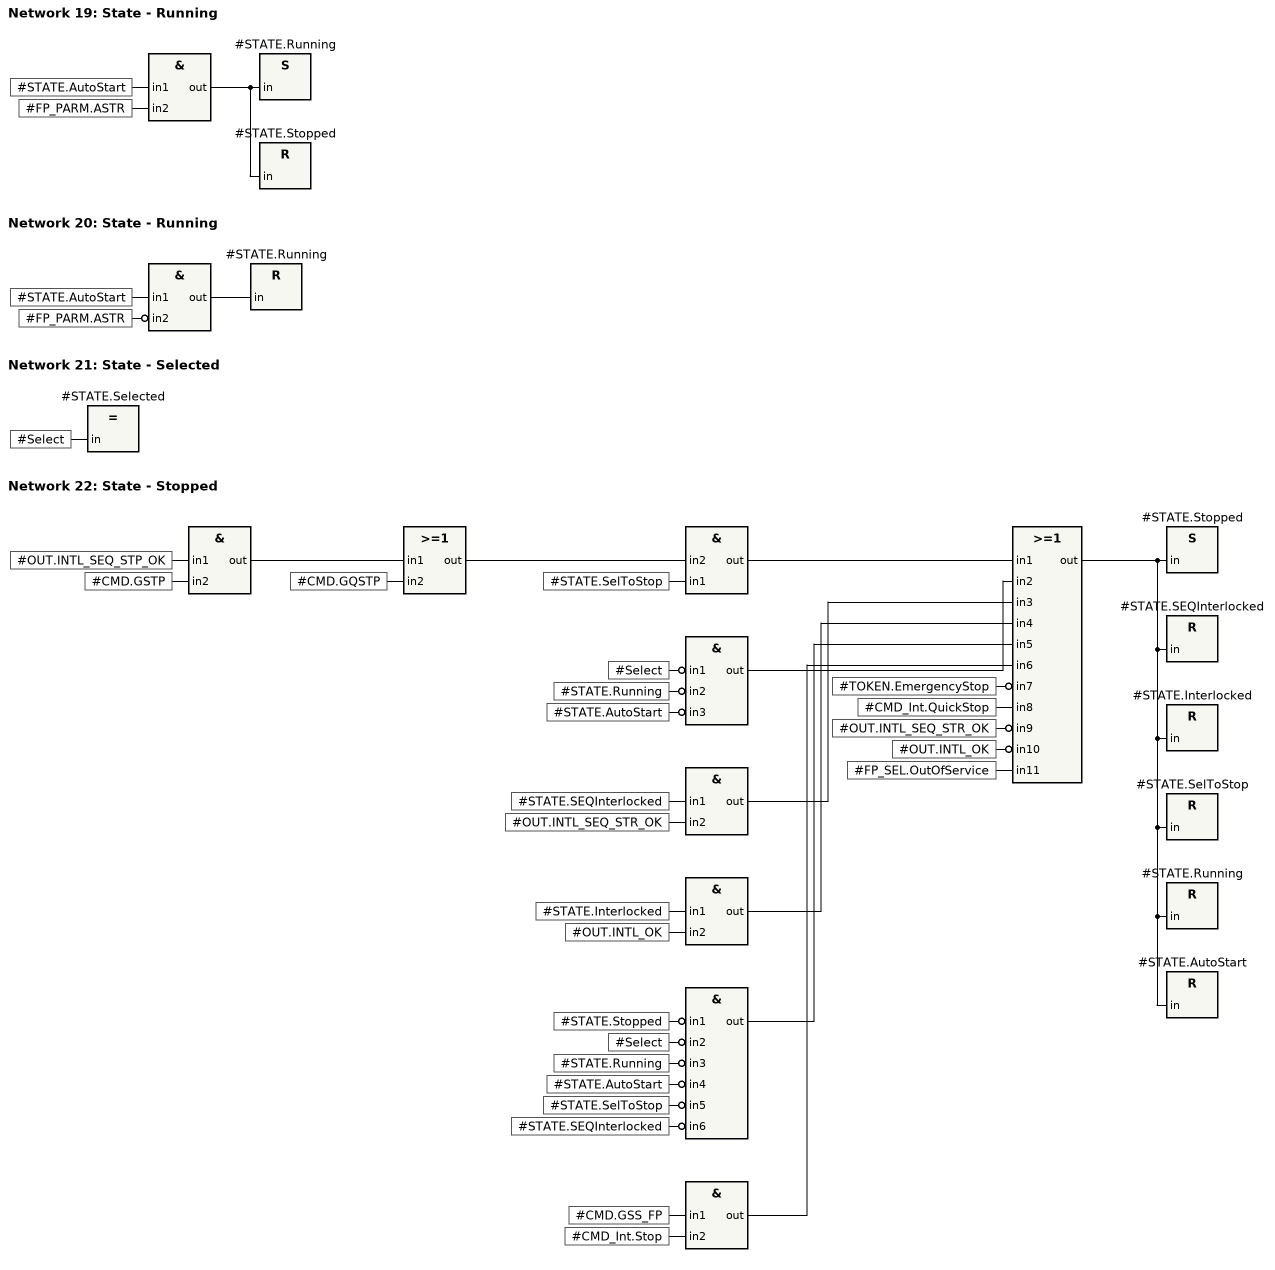
   IF #STATE.AutoStart AND #FP_PARM.ASTR THEN
       #STATE.Running := TRUE;
       #STATE.Stopped := FALSE;
   END_IF;
END_REGION

REGION Network 20: State - Running
   // Build 003-10 Aug 2021- SURAM-IN- State Running Logic unlatched if Auto Start is 
   // 0
   IF #STATE.AutoStart AND NOT #FP_PARM.ASTR THEN #STATE.Running := FALSE; END_IF;
END_REGION

REGION Network 21: State - Selected
   #STATE.Selected := #Select;
END_REGION

REGION Network 22: State - Stopped
   // Build 003-10 Aug 2021- SURAM-IN- State Autostart included along with State Running and State Autostart Unlatch logic added
   #_w1 := (((#OUT.INTL_SEQ_STP_OK AND #CMD.GSTP) OR #CMD.GQSTP) AND #STATE.SelToStop) OR (NOT #Select AND NOT #STATE.Running AND NOT #STATE.AutoStart) OR (#STATE.SEQInterlocked AND #OUT.INTL_SEQ_STR_OK) OR (#STATE.Interlocked AND #OUT.INTL_OK) OR (NOT #STATE.Stopped AND NOT #Select AND NOT #STATE.Running AND NOT #STATE.AutoStart AND NOT #STATE.SelToStop AND NOT #STATE.SEQInterlocked) OR (#CMD.GSS_FP AND #CMD_Int.Stop) OR NOT #TOKEN.EmergencyStop OR #CMD_Int.QuickStop OR NOT #OUT.INTL_SEQ_STR_OK OR NOT #OUT.INTL_OK OR #FP_SEL.OutOfService;
   IF #_w1 THEN
       #STATE.Stopped := TRUE;
       #STATE.SEQInterlocked := FALSE;
       #STATE.Interlocked := FALSE;
       #STATE.SelToStop := FALSE;
       #STATE.Running := FALSE;
       #STATE.AutoStart := FALSE;
   END_IF;
END_REGION

REGION Network 23: State - Single Start
